(* IEC 61131-3 sources: Industry-PLC-LLM/data/PLCBEAD_repo/PLCBEAD_PLCEmbed-main/PLC-BEAD/Source/OpenPLCv2 (part 11) *)

(* ---- CEIL2.ST ---- *)
FUNCTION _REAL_TO_DINT:DINT
  VAR_INPUT
    X :	REAL;
  END_VAR

  IF REAL_TO_DINT(0.5) = DINT#1 THEN
    _REAL_TO_DINT := REAL_TO_DINT(x);
    RETURN;
  END_IF;

  IF X > 0.0 THEN
    _REAL_TO_DINT := REAL_TO_DINT(x+0.5);
  ELSIF X < 0.0 THEN
    _REAL_TO_DINT := REAL_TO_DINT(x-0.5);
  ELSE
    _REAL_TO_DINT := DINT#0;
  END_IF;
END_FUNCTION

FUNCTION CEIL2:DINT

	VAR_INPUT
		X :	REAL;
	END_VAR

	CEIL2 := _REAL_TO_DINT(x);
	IF DINT_TO_REAL(CEIL2) < X THEN
			CEIL2 := CEIL2 + DINT#1;
	END_IF;

END_FUNCTION

PROGRAM program0
  VAR
    LocalVar0 : REAL;
    CEIL5_OUT : DINT;
  END_VAR

  CEIL5_OUT := CEIL2(LocalVar0);
END_PROGRAM

CONFIGURATION Config0

  RESOURCE Res0 ON PLC
    TASK task0(INTERVAL := T#20ms,PRIORITY := 0);
    PROGRAM instance0 WITH task0 : program0;
  END_RESOURCE
END_CONFIGURATION

(* ---- CHECK_PARITY.ST ---- *)
FUNCTION BIT_OF_DWORD : BOOL
  VAR_INPUT
    IN : DWORD;
    N : INT;
  END_VAR

  BIT_OF_DWORD := (SHR(in,N) AND 16#00000001) > 0;
END_FUNCTION

FUNCTION CHECK_PARITY:BOOL

	VAR_INPUT
		IN :	DWORD;
		P :	BOOL;
	END_VAR

	VAR
		in2 :	DWORD;
	END_VAR

	in2:=in;
	check_parity := NOT p;
	WHILE in2 > DWORD#0 DO
		check_parity := check_parity XOR BIT_OF_DWORD(in2,0) XOR BIT_OF_DWORD(in2,1) XOR BIT_OF_DWORD(in2,2) XOR BIT_OF_DWORD(in2,3);
		in2 := SHR(in2,4);
	END_WHILE;

END_FUNCTION

PROGRAM program0
  VAR
    LocalVar0 : DWORD;
    LocalVar1 : BOOL;
    CEIL5_OUT : BOOL;
  END_VAR

  CEIL5_OUT := CHECK_PARITY(LocalVar0, LocalVar1);
END_PROGRAM

CONFIGURATION Config0

  RESOURCE Res0 ON PLC
    TASK task0(INTERVAL := T#20ms,PRIORITY := 0);
    PROGRAM instance0 WITH task0 : program0;
  END_RESOURCE
END_CONFIGURATION

(* ---- CIRCLE_A.ST ---- *)
FUNCTION CIRCLE_A:REAL
	VAR_INPUT
		RX :	REAL;
		AX :	REAL;
	END_VAR

	circle_A := Rx * RX * 8.726646E-3 * Ax;
END_FUNCTION

PROGRAM program0
  VAR
    LocalVar0 : REAL;
	LocalVar1 : REAL;
	LocalOUT  : REAL;
  END_VAR
  	LocalOUT := CIRCLE_A(LocalVar0, LocalVar1);
END_PROGRAM

CONFIGURATION Config0
  RESOURCE Res0 ON PLC
    TASK task0(INTERVAL := T#20ms,PRIORITY := 0);
    PROGRAM instance0 WITH task0 : program0;
  END_RESOURCE
END_CONFIGURATION

(* ---- CIRCLE_C.ST ---- *)
FUNCTION CIRCLE_C:REAL
	VAR_INPUT
		RX :	REAL;
		AX :	REAL;
	END_VAR

	circle_C := 1.7453293E-2 * Rx * Ax;
END_FUNCTION

PROGRAM program0
  VAR
    LocalVar0 : REAL;
	LocalVar1 : REAL;
	LocalOUT  : REAL;
  END_VAR
  	LocalOUT := CIRCLE_C(LocalVar0, LocalVar1);
END_PROGRAM

CONFIGURATION Config0
  RESOURCE Res0 ON PLC
    TASK task0(INTERVAL := T#20ms,PRIORITY := 0);
    PROGRAM instance0 WITH task0 : program0;
  END_RESOURCE
END_CONFIGURATION

(* ---- CIRCLE_SEG.ST ---- *)
FUNCTION CIRCLE_SEG:REAL
	VAR_INPUT
		RX :	REAL;
		HX :	REAL;
	END_VAR

	IF RX > 0.0 THEN
		CIRCLE_SEG := 2.0 * ACOS(1.0 - LIMIT(0.0, HX / RX, 2.0));
		CIRCLE_SEG := (CIRCLE_SEG - SIN(CIRCLE_SEG)) * RX * RX * 0.5;
	END_IF;
END_FUNCTION

PROGRAM program0
  VAR
    LocalVar0 : REAL;
	LocalVar1 : REAL;
	LocalOUT  : REAL;
  END_VAR
  	LocalOUT := CIRCLE_SEG(LocalVar0, LocalVar1);
END_PROGRAM

CONFIGURATION Config0
  RESOURCE Res0 ON PLC
    TASK task0(INTERVAL := T#20ms,PRIORITY := 0);
    PROGRAM instance0 WITH task0 : program0;
  END_RESOURCE
END_CONFIGURATION

(* ---- CMP.ST ---- *)
FUNCTION EXP10 : REAL
  VAR_INPUT
    x : REAL;
  END_VAR

  exp10 := EXP(X * 2.30258509299405);
  (* from OSCAT library; www.oscat.de  *)
END_FUNCTION

FUNCTION FLOOR : INT
  VAR_INPUT
    x : REAL;
  END_VAR

  FLOOR := REAL_TO_INT(X);
  IF INT_TO_REAL(FLOOR) > X THEN
  	floor := floor - 1;
  END_IF;
  (* from OSCAT library; www.oscat.de  *)
END_FUNCTION

FUNCTION CMP:BOOL
	VAR_INPUT
		X :	REAL;
		Y :	REAL;
		N :	INT;
	END_VAR

	VAR
		tmp :	REAL;
	END_VAR

	tmp := ABS(x);
	IF tmp > 0.0 THEN
		tmp := EXP10(INT_TO_REAL(FLOOR(LOG(tmp))-N+1));
	ELSE
		tmp := EXP10(tmp);
	END_IF;
	CMP := ABS(X - Y) < tmp;

END_FUNCTION

PROGRAM program0
  VAR
    LocalVar0 : REAL;
    LocalVar1 : REAL;
	LocalVar2 : INT;
    CEIL5_OUT : BOOL;
  END_VAR

  CEIL5_OUT := CMP(LocalVar0, LocalVar1, LocalVar2);
END_PROGRAM

CONFIGURATION Config0

  RESOURCE Res0 ON PLC
    TASK task0(INTERVAL := T#20ms,PRIORITY := 0);
    PROGRAM instance0 WITH task0 : program0;
  END_RESOURCE
END_CONFIGURATION

(* ---- CONE_V.ST ---- *)
FUNCTION CONE_V:REAL
	VAR_INPUT
		RX :	REAL;
		HX :	REAL;
	END_VAR

	cone_V := 1.047197551 * RX * RX * hx;
END_FUNCTION

PROGRAM program0
  VAR
    LocalVar0 : REAL;
	LocalVar1 : REAL;
	LocalOUT  : REAL;
  END_VAR
  	LocalOUT := CONE_V(LocalVar0, LocalVar1);
END_PROGRAM

CONFIGURATION Config0
  RESOURCE Res0 ON PLC
    TASK task0(INTERVAL := T#20ms,PRIORITY := 0);
    PROGRAM instance0 WITH task0 : program0;
  END_RESOURCE
END_CONFIGURATION

(* ---- COSH.ST ---- *)
FUNCTION COSH:REAL
	VAR_INPUT
		X :	REAL;
	END_VAR

	VAR
		t :	REAL;
	END_VAR

	T := EXP(X);
	COSH := (1.0 / T + T) * 0.5;
END_FUNCTION

PROGRAM program0
  VAR
    LocalVar0 : REAL;
    CEIL5_OUT : REAL;
  END_VAR

  CEIL5_OUT := COSH(LocalVar0);
END_PROGRAM

CONFIGURATION Config0

  RESOURCE Res0 ON PLC
    TASK task0(INTERVAL := T#20ms,PRIORITY := 0);
    PROGRAM instance0 WITH task0 : program0;
  END_RESOURCE
END_CONFIGURATION

(* ---- COTH.ST ---- *)
FUNCTION COTH:REAL

	VAR_INPUT
		X :	REAL;
	END_VAR

	IF X > 20.0 THEN
		COTH :=1.0;
	ELSIF X < -20.0 THEN
		COTH := -1.0;
	ELSE
		COTH := 1.0 + 2.0 / (EXP(X * 2.0) - 1.0);
	END_IF;

END_FUNCTION

PROGRAM program0
	VAR
		X :	REAL;
		OUT : REAL;
	END_VAR

	OUT := COTH(X);

END_PROGRAM

CONFIGURATION Config0

	RESOURCE Res0 ON PLC
		TASK task0(INTERVAL := T#20ms,PRIORITY := 0);
		PROGRAM instance0 WITH task0 : program0;
	END_RESOURCE

END_CONFIGURATION

(* ---- CTRL_IN.ST ---- *)
FUNCTION DEAD_ZONE:REAL

	VAR_INPUT
		X :	REAL;
		L :	REAL;
	END_VAR

	IF ABS(x) > L THEN
		dead_zone := X;
	ELSE
		DEAD_ZONE := 0.0;
	END_IF;

END_FUNCTION

FUNCTION CTRL_IN:REAL
	VAR_INPUT
		SET_POINT :	REAL;
		ACTUAL :	REAL;
		NOISE :	REAL;
	END_VAR
	CTRL_IN := DEAD_ZONE(SET_POINT - ACTUAL, NOISE);
END_FUNCTION

PROGRAM program0
  VAR
    LocalVar0 : REAL;
	LocalVar1 : REAL;
	LocalVar2 : REAL;
	LocalOUT  : REAL;
  END_VAR
  	LocalOUT := CTRL_IN(LocalVar0, LocalVar1, LocalVar2);
END_PROGRAM

CONFIGURATION Config0
  RESOURCE Res0 ON PLC
    TASK task0(INTERVAL := T#20ms,PRIORITY := 0);
    PROGRAM instance0 WITH task0 : program0;
  END_RESOURCE
END_CONFIGURATION

(* ---- D_TRUNC.ST ---- *)
FUNCTION D_TRUNC : DINT
  VAR_INPUT
    x : REAL;
  END_VAR

  D_TRUNC := REAL_TO_DINT(X);
  IF X > 0.0 THEN
  	IF DINT_TO_REAL(D_TRUNC) > X THEN D_TRUNC := D_TRUNC - DINT#1; END_IF;
  ELSE
  	IF DINT_TO_REAL(D_TRUNC) < X THEN D_TRUNC := D_TRUNC + DINT#1; END_IF;
  END_IF;
END_FUNCTION

PROGRAM program0
  VAR
    LocalVar0 : REAL;
    LocalVar1 : DINT;
    CEIL5_OUT : DINT;
  END_VAR

  CEIL5_OUT := D_TRUNC(LocalVar0);
  LocalVar1 := CEIL5_OUT;
END_PROGRAM

CONFIGURATION Config0

  RESOURCE Res0 ON PLC
    TASK task0(INTERVAL := T#20ms,PRIORITY := 0);
    PROGRAM instance0 WITH task0 : program0;
  END_RESOURCE
END_CONFIGURATION

(* ---- DATE_ADD.ST ---- *)
FUNCTION YEAR_OF_DATE:INT
	VAR_INPUT
		IDATE :	UDINT;
	END_VAR

	YEAR_OF_DATE := UDINT_TO_INT((idate+UDINT#43200) / UDINT#31557600 + UDINT#1970);
END_FUNCTION

FUNCTION DAY_OF_WEEK:INT

	VAR_INPUT
		IDATE :	UDINT;
	END_VAR

	DAY_OF_WEEK := UDINT_TO_INT((idate / UDINT#86400 + UDINT#3) MOD UDINT#7) + INT#01;
END_FUNCTION

FUNCTION LEAP_OF_DATE:BOOL

	VAR_INPUT
		IDATE :	UDINT;
	END_VAR

	LEAP_OF_DATE := SHL(UDINT_TO_DWORD((idate + UDINT#43200) / UDINT#31557600), 30) = DWORD#16#80000000;
END_FUNCTION

FUNCTION DAY_OF_YEAR:INT
	VAR_INPUT
		IDATE :	UDINT;
	END_VAR

	DAY_OF_YEAR := UDINT_TO_INT(((idate) / UDINT#86400) MOD UDINT#1461);
	IF DAY_OF_YEAR > 729 THEN
		IF DAY_OF_YEAR > 1095 THEN DAY_OF_YEAR := DAY_OF_YEAR - 1095; ELSE DAY_OF_YEAR := DAY_OF_YEAR - 729; END_IF;
	ELSIF DAY_OF_YEAR > 364 THEN
		DAY_OF_YEAR := DAY_OF_YEAR - 364;
	ELSE
		DAY_OF_YEAR := DAY_OF_YEAR + 1;
	END_IF;
END_FUNCTION

FUNCTION MONTH_OF_DATE:INT

	VAR_INPUT
		IDATE :	UDINT;
	END_VAR

	MONTH_OF_DATE := DAY_OF_YEAR(idate);
	IF MONTH_OF_DATE < 32 THEN
		MONTH_OF_DATE := 1;
	ELSIF LEAP_OF_DATE((IDATE)) THEN
		MONTH_OF_DATE := (MONTH_OF_DATE * 53 + 1668) / 1623;
	ELSE
		MONTH_OF_DATE := (MONTH_OF_DATE * 53 + 1700) / 1620;
	END_IF;
END_FUNCTION

FUNCTION DAY_OF_MONTH:INT
	VAR_INPUT
		IDATE :	UDINT;
	END_VAR

	day_of_month := day_of_year(idate);

	IF leap_of_Date((idate)) THEN
		CASE day_of_month OF
			32..60	:	day_of_month := day_of_month - 31;
			61..91	:	day_of_month := day_of_month - 60;
			92..121 :	day_of_month := day_of_month - 91;
			122..152:	day_of_month := day_of_month - 121;
			153..182:	day_of_month := day_of_month - 152;
			183..213:	day_of_month := day_of_month - 182;
			214..244:	day_of_month := day_of_month - 213;
			245..274:	day_of_month := day_of_month - 244;
			275..305:	day_of_month := day_of_month - 274;
			306..335:	day_of_month := day_of_month - 305;
			336..366:	day_of_month := day_of_month - 335;
		END_CASE;
	ELSE
		CASE day_of_month OF
			32..59	:	day_of_month := day_of_month - 31;
			60..90	:	day_of_month := day_of_month - 59;
			91..120 :	day_of_month := day_of_month - 90;
			121..151:	day_of_month := day_of_month - 120;
			152..181:	day_of_month := day_of_month - 151;
			182..212:	day_of_month := day_of_month - 181;
			213..243:	day_of_month := day_of_month - 212;
			244..273:	day_of_month := day_of_month - 243;
			274..304:	day_of_month := day_of_month - 273;
			305..334:	day_of_month := day_of_month - 304;
			335..365:	day_of_month := day_of_month - 334;
		END_CASE;
	END_IF;
END_FUNCTION

FUNCTION _INT_TO_UDINT:UDINT
	VAR_INPUT
		IN :	INT;
	END_VAR

	_INT_TO_UDINT := DINT_TO_UDINT(INT_TO_DINT(IN));
END_FUNCTION

FUNCTION SET_DATE:UDINT

	VAR_INPUT
		YEAR :	INT;
		MONTH :	INT;
		DAY :	INT;
	END_VAR

	VAR
		count :	INT;
	END_VAR

	IF month > 2 THEN
		count := (month - 1) * 30;
		IF month > 7 THEN
			count := count + DWORD_TO_INT(SHR(DINT_TO_DWORD(INT_TO_DINT(month) - INT_TO_DINT(3)),1));
		ELSE
			count := count + DWORD_TO_INT(SHR(DINT_TO_DWORD(INT_TO_DINT(month) - INT_TO_DINT(4)),1));
		END_IF;
		IF SHL(INT_TO_WORD(year),14) = WORD#0 THEN
			count := count + 1;
		END_IF;
	ELSE
		count := (month - 1) * 31;
	END_IF;
	SET_DATE := (_INT_TO_UDINT(count + day - 1) + DWORD_TO_UDINT(SHR(UDINT_TO_DWORD(_INT_TO_UDINT(year) * UDINT#1461 - UDINT#2878169), 2))) * UDINT#86400;

END_FUNCTION

FUNCTION DATE_ADD:UDINT
	VAR_INPUT
		IDATE :	UDINT;
		D :	INT;
		W :	INT;
		M :	INT;
		Y :	INT;
	END_VAR

	VAR
		mo :	INT;
		yr :	INT;
		dm :	INT;
	END_VAR

	DATE_ADD := IDATE + INT_TO_UDINT(D + W * 7) * UDINT#86400;
	yr := Y + YEAR_OF_DATE(DATE_ADD);
	mo := M + MONTH_OF_DATE(DATE_ADD);
	dm := DAY_OF_MONTH(DATE_ADD);
	WHILE mo > 12 DO
		mo := mo - 12;
		yr := yr + 1;
	END_WHILE;
	WHILE mo < 1 DO
		mo := mo + 12;
		yr := yr - 1;
	END_WHILE;
	DATE_ADD := SET_DATE(yr, mo, dm);
END_FUNCTION

PROGRAM program0
  VAR
    LocalVar0 : UDINT;
	LocalVar1 : INT;
	LocalVar2 : INT;
	LocalVar3 : INT;
	LocalVar4 : INT;
	LocalOUT  : UDINT;
  END_VAR
  	LocalOUT := DATE_ADD(LocalVar0, LocalVar1, LocalVar2, LocalVar3, LocalVar4);
END_PROGRAM

CONFIGURATION Config0
  RESOURCE Res0 ON PLC
    TASK task0(INTERVAL := T#20ms,PRIORITY := 0);
    PROGRAM instance0 WITH task0 : program0;
  END_RESOURCE
END_CONFIGURATION

(* ---- DATE_TO_DT.ST ---- *)
FUNCTION DATE_TO_DT:UDINT
	VAR_INPUT
		IN :	UDINT;
	END_VAR
	DATE_TO_DT := IN;
END_FUNCTION

PROGRAM program0
  VAR
    LocalVar0 : UDINT;
	LocalOUT  : UDINT;
  END_VAR
  	LocalOUT := DATE_TO_DT(LocalVar0);
END_PROGRAM

CONFIGURATION Config0
  RESOURCE Res0 ON PLC
    TASK task0(INTERVAL := T#20ms,PRIORITY := 0);
    PROGRAM instance0 WITH task0 : program0;
  END_RESOURCE
END_CONFIGURATION

(* ---- DATE_TO_DWORD.ST ---- *)
FUNCTION DATE_TO_DWORD2:DWORD
	VAR_INPUT
		IN :	UDINT;
	END_VAR

	DATE_TO_DWORD2 := UDINT_TO_DWORD(IN);
END_FUNCTION

PROGRAM program0
  VAR
    LocalVar0 : UDINT;
	LocalOUT  : DWORD;
  END_VAR
  	LocalOUT := DATE_TO_DWORD2(LocalVar0);
END_PROGRAM

CONFIGURATION Config0
  RESOURCE Res0 ON PLC
    TASK task0(INTERVAL := T#20ms,PRIORITY := 0);
    PROGRAM instance0 WITH task0 : program0;
  END_RESOURCE
END_CONFIGURATION

(* ---- DATE_TO_REAL.ST ---- *)
FUNCTION DATE_TO_REAL2:REAL
	VAR_INPUT
		IN :	UDINT;
	END_VAR

	DATE_TO_REAL2 := UDINT_TO_REAL(IN);
END_FUNCTION

PROGRAM program0
  VAR
    LocalVar0 : UDINT;
	LocalOUT  : REAL;
  END_VAR
  	LocalOUT := DATE_TO_REAL2(LocalVar0);
END_PROGRAM

CONFIGURATION Config0
  RESOURCE Res0 ON PLC
    TASK task0(INTERVAL := T#20ms,PRIORITY := 0);
    PROGRAM instance0 WITH task0 : program0;
  END_RESOURCE
END_CONFIGURATION

(* ---- DATE_TO_UDINT.ST ---- *)
FUNCTION DATE_TO_UDINT2:UDINT
	VAR_INPUT
		IN :	UDINT;
	END_VAR

	DATE_TO_UDINT2 := IN;
END_FUNCTION

PROGRAM program0
  VAR
    LocalVar0 : UDINT;
	LocalOUT  : UDINT;
  END_VAR
  	LocalOUT := DATE_TO_UDINT2(LocalVar0);
END_PROGRAM

CONFIGURATION Config0
  RESOURCE Res0 ON PLC
    TASK task0(INTERVAL := T#20ms,PRIORITY := 0);
    PROGRAM instance0 WITH task0 : program0;
  END_RESOURCE
END_CONFIGURATION

(* ---- DAY_OF_DATE.ST ---- *)
FUNCTION DAY_OF_DATE:DINT
	VAR_INPUT
		IDATE :	UDINT;
	END_VAR

	day_of_date := UDINT_TO_DINT(idate / UDINT#86400);
END_FUNCTION

PROGRAM program0
  VAR
    LocalVar0 : UDINT;
	LocalOUT  : DINT;
  END_VAR
  	LocalOUT := DAY_OF_DATE(LocalVar0);
END_PROGRAM

CONFIGURATION Config0
  RESOURCE Res0 ON PLC
    TASK task0(INTERVAL := T#20ms,PRIORITY := 0);
    PROGRAM instance0 WITH task0 : program0;
  END_RESOURCE
END_CONFIGURATION

(* ---- DAY_OF_MONTH.ST ---- *)
FUNCTION LEAP_OF_DATE:BOOL

	VAR_INPUT
		IDATE :	UDINT;
	END_VAR

	LEAP_OF_DATE := SHL(UDINT_TO_DWORD((idate + UDINT#43200) / UDINT#31557600), 30) = DWORD#16#80000000;

END_FUNCTION

FUNCTION DAY_OF_YEAR:INT
	VAR_INPUT
		IDATE :	DATE;
	END_VAR

	DAY_OF_YEAR := UDINT_TO_INT((DATE_TO_UDINT(idate) / UDINT#86400) MOD UDINT#1461);
	IF DAY_OF_YEAR > 729 THEN
		IF DAY_OF_YEAR > 1095 THEN DAY_OF_YEAR := DAY_OF_YEAR - 1095; ELSE DAY_OF_YEAR := DAY_OF_YEAR - 729; END_IF;
	ELSIF DAY_OF_YEAR > 364 THEN
		DAY_OF_YEAR := DAY_OF_YEAR - 364;
	ELSE
		DAY_OF_YEAR := DAY_OF_YEAR + 1;
	END_IF;
END_FUNCTION

FUNCTION DAY_OF_MONTH:INT
	VAR_INPUT
		IDATE :	DATE;
	END_VAR

	day_of_month := day_of_year(idate);

	IF leap_of_Date(DATE_TO_UDINT(idate)) THEN
		CASE day_of_month OF
			32..60	:	day_of_month := day_of_month - 31;
			61..91	:	day_of_month := day_of_month - 60;
			92..121 :	day_of_month := day_of_month - 91;
			122..152:	day_of_month := day_of_month - 121;
			153..182:	day_of_month := day_of_month - 152;
			183..213:	day_of_month := day_of_month - 182;
			214..244:	day_of_month := day_of_month - 213;
			245..274:	day_of_month := day_of_month - 244;
			275..305:	day_of_month := day_of_month - 274;
			306..335:	day_of_month := day_of_month - 305;
			336..366:	day_of_month := day_of_month - 335;
		END_CASE;
	ELSE
		CASE day_of_month OF
			32..59	:	day_of_month := day_of_month - 31;
			60..90	:	day_of_month := day_of_month - 59;
			91..120 :	day_of_month := day_of_month - 90;
			121..151:	day_of_month := day_of_month - 120;
			152..181:	day_of_month := day_of_month - 151;
			182..212:	day_of_month := day_of_month - 181;
			213..243:	day_of_month := day_of_month - 212;
			244..273:	day_of_month := day_of_month - 243;
			274..304:	day_of_month := day_of_month - 273;
			305..334:	day_of_month := day_of_month - 304;
			335..365:	day_of_month := day_of_month - 334;
		END_CASE;
	END_IF;

END_FUNCTION

PROGRAM program0
  VAR
    LocalVar0 : DATE;
	LocalOUT  : INT;
  END_VAR
  	LocalOUT := DAY_OF_MONTH(LocalVar0);
END_PROGRAM

CONFIGURATION Config0
  RESOURCE Res0 ON PLC
    TASK task0(INTERVAL := T#20ms,PRIORITY := 0);
    PROGRAM instance0 WITH task0 : program0;
  END_RESOURCE
END_CONFIGURATION

(* ---- DAY_OF_WEEK.ST ---- *)
FUNCTION DAY_OF_WEEK:INT
  VAR_INPUT
    IDATE :	UDINT;
  END_VAR

  DAY_OF_WEEK := UDINT_TO_INT((idate / UDINT#86400 + UDINT#3) MOD UDINT#7) + INT#01;
END_FUNCTION

PROGRAM program0
  VAR
    LocalVar0 : UDINT;
	LocalOUT  : INT;
  END_VAR
  	LocalOUT := DAY_OF_WEEK(LocalVar0);
END_PROGRAM

CONFIGURATION Config0
  RESOURCE Res0 ON PLC
    TASK task0(INTERVAL := T#20ms,PRIORITY := 0);
    PROGRAM instance0 WITH task0 : program0;
  END_RESOURCE
END_CONFIGURATION

(* ---- DAY_OF_YEAR.ST ---- *)
FUNCTION DAY_OF_YEAR:INT
	VAR_INPUT
		IDATE :	DATE;
	END_VAR

	DAY_OF_YEAR := UDINT_TO_INT((DATE_TO_UDINT(idate) / UDINT#86400) MOD UDINT#1461);
	IF DAY_OF_YEAR > 729 THEN
		IF DAY_OF_YEAR > 1095 THEN DAY_OF_YEAR := DAY_OF_YEAR - 1095; ELSE DAY_OF_YEAR := DAY_OF_YEAR - 729; END_IF;
	ELSIF DAY_OF_YEAR > 364 THEN
		DAY_OF_YEAR := DAY_OF_YEAR - 364;
	ELSE
		DAY_OF_YEAR := DAY_OF_YEAR + 1;
	END_IF;
END_FUNCTION

PROGRAM program0
  VAR
    LocalVar0 : DATE;
	LocalOUT  : INT;
  END_VAR
  	LocalOUT := DAY_OF_YEAR(LocalVar0);
END_PROGRAM

CONFIGURATION Config0
  RESOURCE Res0 ON PLC
    TASK task0(INTERVAL := T#20ms,PRIORITY := 0);
    PROGRAM instance0 WITH task0 : program0;
  END_RESOURCE
END_CONFIGURATION

(* ---- DAYS_DELTA.ST ---- *)
FUNCTION DAYS_DELTA:DINT
	VAR_INPUT
		DATE_1 :	UDINT;
		DATE_2 :	UDINT;
	END_VAR
	IF DATE_1 > DATE_2 THEN
		DAYS_DELTA := - UDINT_TO_DINT((date_1 - date_2) / UDINT#86400);
	ELSE
		DAYS_DELTA :=   UDINT_TO_DINT((date_2 - date_1) / UDINT#86400);
	END_IF;
END_FUNCTION

PROGRAM program0
  VAR
    LocalVar0 : UDINT;
	LocalVar1 : UDINT;
	LocalOUT  : DINT;
  END_VAR
  	LocalOUT := DAYS_DELTA(LocalVar0, LocalVar1);
END_PROGRAM

CONFIGURATION Config0
  RESOURCE Res0 ON PLC
    TASK task0(INTERVAL := T#20ms,PRIORITY := 0);
    PROGRAM instance0 WITH task0 : program0;
  END_RESOURCE
END_CONFIGURATION

(* ---- DAYS_IN_MONTH.ST ---- *)
FUNCTION DAY_OF_YEAR:INT
	VAR_INPUT
		IDATE :	UDINT;
	END_VAR

	DAY_OF_YEAR := UDINT_TO_INT(((idate) / UDINT#86400) MOD UDINT#1461);
	IF DAY_OF_YEAR > 729 THEN
		IF DAY_OF_YEAR > 1095 THEN DAY_OF_YEAR := DAY_OF_YEAR - 1095; ELSE DAY_OF_YEAR := DAY_OF_YEAR - 729; END_IF;
	ELSIF DAY_OF_YEAR > 364 THEN
		DAY_OF_YEAR := DAY_OF_YEAR - 364;
	ELSE
		DAY_OF_YEAR := DAY_OF_YEAR + 1;
	END_IF;
END_FUNCTION

FUNCTION LEAP_OF_DATE:BOOL

	VAR_INPUT
		IDATE :	UDINT;
	END_VAR

	LEAP_OF_DATE := SHL(UDINT_TO_DWORD((idate + UDINT#43200) / UDINT#31557600), 30) = DWORD#16#80000000;
END_FUNCTION

FUNCTION DAYS_IN_MONTH:INT

	VAR_INPUT
		IDATE :	UDINT;
	END_VAR

	DAYS_IN_MONTH := DAY_OF_YEAR(IDATE);
	IF LEAP_OF_DATE(IDATE) THEN
		CASE DAYS_IN_MONTH OF
			32..60	:	DAYS_IN_MONTH := 29;
			92..121 :	DAYS_IN_MONTH := 30;
			153..182:	DAYS_IN_MONTH := 30;
			245..274:	DAYS_IN_MONTH := 30;
			306..335:	DAYS_IN_MONTH := 30;
		ELSE
			DAYS_IN_MONTH := 31;
		END_CASE;
	ELSE
		CASE DAYS_IN_MONTH OF
			32..59	:	DAYS_IN_MONTH := 28;
			91..120 :	DAYS_IN_MONTH := 30;
			152..181:	DAYS_IN_MONTH := 30;
			244..273:	DAYS_IN_MONTH := 30;
			305..334:	DAYS_IN_MONTH := 30;
		ELSE
			DAYS_IN_MONTH := 31;
		END_CASE;
	END_IF;

END_FUNCTION

PROGRAM program0
  VAR
    LocalVar0 : UDINT;
	LocalOUT  : INT;
  END_VAR
  	LocalOUT := DAYS_IN_MONTH(LocalVar0);
END_PROGRAM

CONFIGURATION Config0
  RESOURCE Res0 ON PLC
    TASK task0(INTERVAL := T#20ms,PRIORITY := 0);
    PROGRAM instance0 WITH task0 : program0;
  END_RESOURCE
END_CONFIGURATION

(* ---- DAYS_IN_YEAR.ST ---- *)
FUNCTION LEAP_OF_DATE:BOOL

	VAR_INPUT
		IDATE :	UDINT;
	END_VAR

	LEAP_OF_DATE := SHL(UDINT_TO_DWORD((idate + UDINT#43200) / UDINT#31557600), 30) = DWORD#16#80000000;
END_FUNCTION

FUNCTION DAYS_IN_YEAR:INT
	VAR_INPUT
		IDATE :	UDINT;
	END_VAR

	IF LEAP_OF_DATE(IDATE) THEN
		DAYS_IN_YEAR := 366;
	ELSE
		DAYS_IN_YEAR := 365;
	END_IF;
END_FUNCTION

PROGRAM program0
  VAR
    LocalVar0 : UDINT;
	LocalOUT  : INT;
  END_VAR
  	LocalOUT := DAYS_IN_YEAR(LocalVar0);
END_PROGRAM

CONFIGURATION Config0
  RESOURCE Res0 ON PLC
    TASK task0(INTERVAL := T#20ms,PRIORITY := 0);
    PROGRAM instance0 WITH task0 : program0;
  END_RESOURCE
END_CONFIGURATION

(* ---- DEAD_BAND.ST ---- *)
FUNCTION DEAD_BAND:REAL

	VAR_INPUT
		X :	REAL;
		L :	REAL;
	END_VAR

	IF X > L THEN
		DEAD_BAND := X - L;
	ELSIF X < -L THEN
		DEAD_BAND := X + L;
	ELSE
		DEAD_BAND := 0.0;
	END_IF;

END_FUNCTION

PROGRAM program0
  VAR
    LocalVar0 : REAL;
	LocalVar1 : REAL;
	LocalOUT  : REAL;
  END_VAR
  	LocalOUT := DEAD_BAND(LocalVar0, LocalVar1);
END_PROGRAM

CONFIGURATION Config0
  RESOURCE Res0 ON PLC
    TASK task0(INTERVAL := T#20ms,PRIORITY := 0);
    PROGRAM instance0 WITH task0 : program0;
  END_RESOURCE
END_CONFIGURATION

(* ---- DEAD_ZONE.ST ---- *)
FUNCTION DEAD_ZONE:REAL

	VAR_INPUT
		X :	REAL;
		L :	REAL;
	END_VAR

	IF ABS(x) > L THEN
		dead_zone := X;
	ELSE
		DEAD_ZONE := 0.0;
	END_IF;

END_FUNCTION

PROGRAM program0
  VAR
    LocalVar0 : REAL;
	LocalVar1 : REAL;
	LocalOUT  : REAL;
  END_VAR
  	LocalOUT := DEAD_ZONE(LocalVar0, LocalVar1);
END_PROGRAM

CONFIGURATION Config0
  RESOURCE Res0 ON PLC
    TASK task0(INTERVAL := T#20ms,PRIORITY := 0);
    PROGRAM instance0 WITH task0 : program0;
  END_RESOURCE
END_CONFIGURATION

(* ---- DEC1.ST ---- *)
FUNCTION DEC1:INT

	VAR_INPUT
		X :	INT;
		N :	INT;
	END_VAR

	IF X = 0 THEN
		DEC1 := N - 1;
	ELSE
		DEC1 := X - 1;
	END_IF;

END_FUNCTION

PROGRAM program0
  VAR
    LocalVar0 : INT;
	LocalVar1 : INT;
	LocalOUT  : INT;
  END_VAR
  	LocalOUT := DEC1(LocalVar0, LocalVar1);
END_PROGRAM

CONFIGURATION Config0
  RESOURCE Res0 ON PLC
    TASK task0(INTERVAL := T#20ms,PRIORITY := 0);
    PROGRAM instance0 WITH task0 : program0;
  END_RESOURCE
END_CONFIGURATION

(* ---- DEG.ST ---- *)
FUNCTION FLOOR2 : DINT
	VAR_INPUT
		x : REAL;
	END_VAR

	FLOOR2 := REAL_TO_DINT(X);
	IF DINT_TO_REAL(FLOOR2) > X THEN
		FLOOR2 := FLOOR2 - DINT#1;
	END_IF;

END_FUNCTION

FUNCTION MODR:REAL

	VAR_INPUT
		IN :	REAL;
		DIVI :	REAL;
	END_VAR

	IF divi = 0.0 THEN
		MODR := 0.0;
	ELSE
		MODR := in - DINT_TO_REAL(FLOOR2(in / divi)) * divi;
	END_IF;

END_FUNCTION

FUNCTION DEG:REAL

	VAR_INPUT
		RAD :	REAL;
	END_VAR

	DEG := MODR(57.29577951308232 * RAD, 360.0);

END_FUNCTION

PROGRAM program0

	VAR
		RAD :	REAL;
		CEIL5_OUT : REAL;
	END_VAR

	CEIL5_OUT := DEG(RAD);

END_PROGRAM

CONFIGURATION Config0

	RESOURCE Res0 ON PLC
		TASK task0(INTERVAL := T#20ms,PRIORITY := 0);
		PROGRAM instance0 WITH task0 : program0;
	END_RESOURCE

END_CONFIGURATION

(* ---- DEW_CON.ST ---- *)
FUNCTION SDD:REAL

	VAR_INPUT
		T :	REAL;
		ICE :	BOOL;
	END_VAR

	IF ice THEN
		SDD := 611.153 * EXP(22.4433 * T / (272.186 + T));
	ELSE
		SDD := 611.213 * EXP(17.5043 * T / (241.2 + T));
	END_IF;

END_FUNCTION

FUNCTION DEW_CON:REAL

	VAR_INPUT
		RH :	REAL;
		T :	REAL;
	END_VAR

	IF RH > 0.0 AND T > -50.0 THEN
		DEW_CON := 2.166824303E-2 * RH * SDD(T,FALSE)  / (T - -273.15);
	ELSE
		DEW_CON := 0.0;
	END_IF;

END_FUNCTION

PROGRAM program0
  VAR
    RH :	REAL;
	T :	REAL;
    CEIL5_OUT : REAL;
  END_VAR

  CEIL5_OUT := DEW_CON(RH, T);
END_PROGRAM

CONFIGURATION Config0

  RESOURCE Res0 ON PLC
    TASK task0(INTERVAL := T#20ms,PRIORITY := 0);
    PROGRAM instance0 WITH task0 : program0;
  END_RESOURCE
END_CONFIGURATION

(* ---- DEW_RH.ST ---- *)
FUNCTION SDD:REAL

	VAR_INPUT
		T :	REAL;
		ICE :	BOOL;
	END_VAR

	IF ice THEN
		SDD := 611.153 * EXP(22.4433 * T / (272.186 + T));
	ELSE
		SDD := 611.213 * EXP(17.5043 * T / (241.2 + T));
	END_IF;

END_FUNCTION

FUNCTION DEW_CON:REAL

	VAR_INPUT
		RH :	REAL;
		T :	REAL;
	END_VAR

	IF RH > 0.0 AND T > -50.0 THEN
		DEW_CON := 2.166824303E-2 * RH * SDD(T,FALSE)  / (T - -273.15);
	ELSE
		DEW_CON := 0.0;
	END_IF;

END_FUNCTION

FUNCTION DEW_RH:REAL

	VAR_INPUT
		VC :	REAL;
		T :	REAL;
	END_VAR

	DEW_RH := LIMIT(0.0, VC / DEW_CON(1.0, T), 100.0);

END_FUNCTION

PROGRAM program0
	VAR
		VC :	REAL;
		T :	REAL;
		CEIL5_OUT : REAL;
	END_VAR

  	CEIL5_OUT := DEW_RH(VC, T);
END_PROGRAM

CONFIGURATION Config0

  RESOURCE Res0 ON PLC
    TASK task0(INTERVAL := T#20ms,PRIORITY := 0);
    PROGRAM instance0 WITH task0 : program0;
  END_RESOURCE
END_CONFIGURATION

(* ---- DEW_TEMP.ST ---- *)
FUNCTION EXP10 : REAL
  VAR_INPUT
    x : REAL;
  END_VAR

  exp10 := EXP(X * 2.30258509299405);
  (* from OSCAT library; www.oscat.de  *)
END_FUNCTION

FUNCTION DEW_TEMP:REAL

VAR_INPUT
	RH :	REAL;
	T :	REAL;
END_VAR

	VAR
		V :	REAL;
	END_VAR

	IF rh > 0.0 THEN

		V := LOG(RH * 0.01 * EXP10((7.5*T) / (237.3+T)));
		DEW_TEMP := 237.3*V / (7.5-V);
	ELSE
		DEW_TEMP:= -273.15;
	END_IF;

END_FUNCTION

PROGRAM program0
	VAR
		RH :	REAL;
		T :	REAL;
		CEIL5_OUT : REAL;
	END_VAR

  	CEIL5_OUT := DEW_TEMP(RH, T);
END_PROGRAM

CONFIGURATION Config0

  RESOURCE Res0 ON PLC
    TASK task0(INTERVAL := T#20ms,PRIORITY := 0);
    PROGRAM instance0 WITH task0 : program0;
  END_RESOURCE
END_CONFIGURATION

(* ---- DIFFER.ST ---- *)
FUNCTION DIFFER:BOOL
	VAR_INPUT
		IN1 :	REAL;
		IN2 :	REAL;
		X :	REAL;
	END_VAR

	DIFFER := ABS(in1 - in2) > X;
END_FUNCTION

PROGRAM program0
  VAR
    LocalVar0 : REAL;
	LocalVar1 : REAL;
	LocalVar2 : REAL;
	LocalOUT  : BOOL;
  END_VAR
  	LocalOUT := DIFFER(LocalVar0, LocalVar1, LocalVar2);
END_PROGRAM

CONFIGURATION Config0
  RESOURCE Res0 ON PLC
    TASK task0(INTERVAL := T#20ms,PRIORITY := 0);
    PROGRAM instance0 WITH task0 : program0;
  END_RESOURCE
END_CONFIGURATION

(* ---- DST.ST ---- *)
FUNCTION _INT_TO_UDINT:UDINT
	VAR_INPUT
		IN :	INT;
	END_VAR

	_INT_TO_UDINT := DINT_TO_UDINT(INT_TO_DINT(IN));
END_FUNCTION

FUNCTION YEAR_OF_DATE:INT
	VAR_INPUT
		IDATE :	UDINT;
	END_VAR

	YEAR_OF_DATE := UDINT_TO_INT((idate+UDINT#43200) / UDINT#31557600 + UDINT#1970);
END_FUNCTION

FUNCTION DT_TO_DATE2:UDINT

	VAR_INPUT
		IN :	UDINT;
	END_VAR

	DT_TO_DATE2 := (IN / UDINT#86400) * UDINT#86400;
END_FUNCTION

FUNCTION SET_DATE:UDINT

	VAR_INPUT
		YEAR :	INT;
		MONTH :	INT;
		DAY :	INT;
	END_VAR

	VAR
		count :	INT;
	END_VAR

	IF month > 2 THEN
		count := (month - 1) * 30;
		IF month > 7 THEN
			count := count + DWORD_TO_INT(SHR(DINT_TO_DWORD(INT_TO_DINT(month) - INT_TO_DINT(3)),1));
		ELSE
			count := count + DWORD_TO_INT(SHR(DINT_TO_DWORD(INT_TO_DINT(month) - INT_TO_DINT(4)),1));
		END_IF;
		IF SHL(INT_TO_WORD(year),14) = WORD#0 THEN
			count := count + 1;
		END_IF;
	ELSE
		count := (month - 1) * 31;
	END_IF;
	SET_DATE := (_INT_TO_UDINT(count + day - 1) + DWORD_TO_UDINT(SHR(UDINT_TO_DWORD(_INT_TO_UDINT(year) * UDINT#1461 - UDINT#2878169), 2))) * UDINT#86400;

END_FUNCTION

FUNCTION SET_DT:UDINT

	VAR_INPUT
		YEAR :	INT;
		MONTH :	INT;
		DAY :	INT;
		HOUR :	INT;
		MINUTE :	INT;
		SECOND :	INT;
	END_VAR

	SET_DT := SET_DATE(YEAR, MONTH, DAY) + _INT_TO_UDINT(SECOND) + _INT_TO_UDINT(MINUTE) * UDINT#60 + _INT_TO_UDINT(HOUR) * UDINT#3600;

END_FUNCTION

FUNCTION DST:BOOL
	VAR_INPUT
		UTC :	UDINT;
	END_VAR

	VAR
		yr :	INT;
		yr4 :	UDINT;
		ltc :	UDINT;
		idate :	UDINT;
	END_VAR

	yr := YEAR_OF_DATE(DT_TO_DATE2(UTC));
	ltc := UTC;
	idate := SET_DT(yr, 3, 31, 1, 0, 0);
	yr4 := DWORD_TO_UDINT(SHR(INT_TO_DWORD(5 * yr), 2)) + UDINT#1;
	DST := (idate - ((yr4 + UDINT#3) MOD UDINT#7) * UDINT#86400 <= ltc) AND (idate + (UDINT#214 - (yr4) MOD UDINT#7) * UDINT#86400 > ltc);
END_FUNCTION

PROGRAM program0
	VAR
		UTC :	UDINT;
		CEIL5_OUT : BOOL;
	END_VAR

  CEIL5_OUT := DST(UTC);

END_PROGRAM

CONFIGURATION Config0
	RESOURCE Res0 ON PLC
		TASK task0(INTERVAL := T#20ms,PRIORITY := 0);
		PROGRAM instance0 WITH task0 : program0;
	END_RESOURCE
END_CONFIGURATION

(* ---- DT_TO_TOD.ST ---- *)
FUNCTION DT_TO_TOD2:UDINT
	VAR_INPUT
		IN :	UDINT;
	END_VAR

	DT_TO_TOD2 := (IN MOD UDINT#86400) * UDINT#1000;
END_FUNCTION

PROGRAM program0
  VAR
    LocalVar0 : UDINT;
	LocalOUT  : UDINT;
  END_VAR
  	LocalOUT := DT_TO_TOD2(LocalVar0);
END_PROGRAM

CONFIGURATION Config0
  RESOURCE Res0 ON PLC
    TASK task0(INTERVAL := T#20ms,PRIORITY := 0);
    PROGRAM instance0 WITH task0 : program0;
  END_RESOURCE
END_CONFIGURATION

(* ---- DWORD_OF_BYTE.ST ---- *)
FUNCTION DWORD_OF_BYTE:DWORD
	VAR_INPUT
		B3 :	BYTE;
		B2 :	BYTE;
		B1 :	BYTE;
		B0 :	BYTE;
	END_VAR

	DWORD_OF_BYTE := SHL(SHL(SHL(BYTE_TO_DWORD(B3),8) OR BYTE_TO_DWORD(B2),8) OR BYTE_TO_DWORD(B1),8) OR BYTE_TO_DWORD(B0);

END_FUNCTION

PROGRAM program0
  VAR
    LocalVar0 : BYTE;
	LocalVar1 : BYTE;
	LocalVar2 : BYTE;
	LocalVar3 : BYTE;
	LocalOUT  : DWORD;
  END_VAR
  	LocalOUT := DWORD_OF_BYTE(LocalVar0, LocalVar1, LocalVar2, LocalVar3);
END_PROGRAM

CONFIGURATION Config0
  RESOURCE Res0 ON PLC
    TASK task0(INTERVAL := T#20ms,PRIORITY := 0);
    PROGRAM instance0 WITH task0 : program0;
  END_RESOURCE
END_CONFIGURATION

(* ---- DWORD_OF_WORD.ST ---- *)
FUNCTION DWORD_OF_WORD:DWORD

	VAR_INPUT
		W1 :	WORD;
		W0 :	WORD;
	END_VAR

	DWORD_OF_WORD := SHL(WORD_TO_DWORD(W1),16) OR WORD_TO_DWORD(W0);

END_FUNCTION

PROGRAM program0
  VAR
    LocalVar0 : WORD;
	LocalVar1 : WORD;
	LocalOUT  : DWORD;
  END_VAR
  	LocalOUT := DWORD_OF_WORD(LocalVar0, LocalVar1);
END_PROGRAM

CONFIGURATION Config0
  RESOURCE Res0 ON PLC
    TASK task0(INTERVAL := T#20ms,PRIORITY := 0);
    PROGRAM instance0 WITH task0 : program0;
  END_RESOURCE
END_CONFIGURATION

(* ---- DWORD_TO_DATE.ST ---- *)
FUNCTION DWORD_TO_DATE2:UDINT
	VAR_INPUT
		IN :	DWORD;
	END_VAR
	DWORD_TO_DATE2 := DWORD_TO_UDINT(IN);
END_FUNCTION

PROGRAM program0
  VAR
    LocalVar0 : DWORD;
	LocalOUT  : UDINT;
  END_VAR
  	LocalOUT := DWORD_TO_DATE2(LocalVar0);
END_PROGRAM

CONFIGURATION Config0
  RESOURCE Res0 ON PLC
    TASK task0(INTERVAL := T#20ms,PRIORITY := 0);
    PROGRAM instance0 WITH task0 : program0;
  END_RESOURCE
END_CONFIGURATION

(* ---- DWORD_TO_DT.ST ---- *)
FUNCTION DWORD_TO_DT2:UDINT

	VAR_INPUT
		IN :	DWORD;
	END_VAR

	DWORD_TO_DT2 := DWORD_TO_UDINT(IN);
END_FUNCTION

PROGRAM program0
  VAR
    LocalVar0 : DWORD;
	LocalOUT  : UDINT;
  END_VAR
  	LocalOUT := DWORD_TO_DT2(LocalVar0);
END_PROGRAM

CONFIGURATION Config0
  RESOURCE Res0 ON PLC
    TASK task0(INTERVAL := T#20ms,PRIORITY := 0);
    PROGRAM instance0 WITH task0 : program0;
  END_RESOURCE
END_CONFIGURATION

(* ---- DWORD_TO_TIME.ST ---- *)
FUNCTION DWORD_TO_TIME2:TIME
	VAR_INPUT
		X :	DWORD;
	END_VAR
	DWORD_TO_TIME2 := DINT_TO_TIME(DWORD_TO_DINT(X));
END_FUNCTION

PROGRAM program0
  VAR
    LocalVar0 : DWORD;
	  LocalOUT  : TIME;
  END_VAR
  	LocalOUT := DWORD_TO_TIME2(LocalVar0);
END_PROGRAM

CONFIGURATION Config0
  RESOURCE Res0 ON PLC
    TASK task0(INTERVAL := T#20ms,PRIORITY := 0);
    PROGRAM instance0 WITH task0 : program0;
  END_RESOURCE
END_CONFIGURATION

(* ---- DWORD_TO_TOD.ST ---- *)
FUNCTION DWORD_TO_TOD2:UDINT
	VAR_INPUT
		IN :	DWORD;
	END_VAR
	DWORD_TO_TOD2 := DWORD_TO_UDINT(IN);
END_FUNCTION

PROGRAM program0
  VAR
    LocalVar0 : DWORD;
	  LocalOUT  : UDINT;
  END_VAR
  	LocalOUT := DWORD_TO_TOD2(LocalVar0);
END_PROGRAM

CONFIGURATION Config0
  RESOURCE Res0 ON PLC
    TASK task0(INTERVAL := T#20ms,PRIORITY := 0);
    PROGRAM instance0 WITH task0 : program0;
  END_RESOURCE
END_CONFIGURATION

(* ---- EASTER.ST ---- *)
FUNCTION _INT_TO_UDINT:UDINT
	VAR_INPUT
		IN :	INT;
	END_VAR

	_INT_TO_UDINT := DINT_TO_UDINT(INT_TO_DINT(IN));
END_FUNCTION

FUNCTION SET_DATE:UDINT

	VAR_INPUT
		YEAR :	INT;
		MONTH :	INT;
		DAY :	INT;
	END_VAR

	VAR
		count :	INT;
	END_VAR

	IF month > 2 THEN
		count := (month - 1) * 30;
		IF month > 7 THEN
			count := count + DWORD_TO_INT(SHR(DINT_TO_DWORD(INT_TO_DINT(month) - INT_TO_DINT(3)),1));
		ELSE
			count := count + DWORD_TO_INT(SHR(DINT_TO_DWORD(INT_TO_DINT(month) - INT_TO_DINT(4)),1));
		END_IF;
		IF SHL(INT_TO_WORD(year),14) = WORD#0 THEN
			count := count + 1;
		END_IF;
	ELSE
		count := (month - 1) * 31;
	END_IF;
	SET_DATE := (_INT_TO_UDINT(count + day - 1) + DWORD_TO_UDINT(SHR(UDINT_TO_DWORD(_INT_TO_UDINT(year) * UDINT#1461 - UDINT#2878169), 2))) * UDINT#86400;

END_FUNCTION

FUNCTION EASTER:UDINT
	VAR_INPUT
		YEAR :	INT;
	END_VAR

	VAR
		b :	INT;
		c :	INT;
		oday :	INT;
	END_VAR

	b := (204 - 11 * (year MOD 19)) MOD 30;
	IF b > 27 THEN b := b - 1; END_IF;
	c := (year + WORD_TO_INT(SHR(INT_TO_WORD(year),2)) + b - 13) MOD 7;
	oday := 28 + b - c;
	IF oday > 33 THEN
		easter := set_Date(year, 4, oday - 31);
	ELSE
		easter := set_Date(year, 3, oday);
	END_IF;
END_FUNCTION

PROGRAM program0
  VAR
    LocalVar0 : INT;
	LocalOUT  : UDINT;
  END_VAR
  	LocalOUT := EASTER(LocalVar0);
END_PROGRAM

CONFIGURATION Config0
  RESOURCE Res0 ON PLC
    TASK task0(INTERVAL := T#20ms,PRIORITY := 0);
    PROGRAM instance0 WITH task0 : program0;
  END_RESOURCE
END_CONFIGURATION

(* ---- ELLIPSE_A.ST ---- *)
FUNCTION ELLIPSE_A:REAL
	VAR_INPUT
		R1 :	REAL;
		R2 :	REAL;
	END_VAR

	ellipse_A := 3.14159265358979323846264338327950288 * R1 * R2;

END_FUNCTION

PROGRAM program0
  VAR
    LocalVar0 : REAL;
	LocalVar1 : REAL;
	  LocalOUT  : REAL;
  END_VAR
  	LocalOUT := ELLIPSE_A(LocalVar0, LocalVar1);
END_PROGRAM

CONFIGURATION Config0
  RESOURCE Res0 ON PLC
    TASK task0(INTERVAL := T#20ms,PRIORITY := 0);
    PROGRAM instance0 WITH task0 : program0;
  END_RESOURCE
END_CONFIGURATION

(* ---- ELLIPSE_C.ST ---- *)
FUNCTION ELLIPSE_C:REAL

VAR_INPUT
	R1 :	REAL;
	R2 :	REAL;
END_VAR

ELLIPSE_C := 3.14159265358979323846264338327950288 * (3.0 * (R1+R2) - SQRT((3.0 * r1 + R2) * (3.0 * r2 + r1)));

END_FUNCTION

PROGRAM program0
  VAR
    LocalVar0 : REAL;
	LocalVar1 : REAL;
	  LocalOUT  : REAL;
  END_VAR
  	LocalOUT := ELLIPSE_C(LocalVar0, LocalVar1);
END_PROGRAM

CONFIGURATION Config0
  RESOURCE Res0 ON PLC
    TASK task0(INTERVAL := T#20ms,PRIORITY := 0);
    PROGRAM instance0 WITH task0 : program0;
  END_RESOURCE
END_CONFIGURATION

(* ---- ERF.ST ---- *)
FUNCTION SGN : INT
  VAR_INPUT
    x : REAL;
  END_VAR

  IF X > 0.0 THEN
  	sgn := 1;
  ELSIF X < 0.0 THEN
  	sgn := -1;
  ELSE
  	sgn := 0;
  END_IF;
END_FUNCTION

FUNCTION ERF:REAL

	VAR_INPUT
		X :	REAL;
	END_VAR

	VAR
		x2 :	REAL;
		ax2 :	REAL;
	END_VAR

	x2 := X*X;
	ax2 := 0.147 * x2 + 1.0;
	ERF := SQRT(1.0 - EXP(-X2 * ((0.27323954473516 + aX2)/(ax2)))) * INT_TO_REAL(SGN(x));

END_FUNCTION

PROGRAM program0
  VAR
    LocalVar0 : REAL;
	  LocalOUT  : REAL;
  END_VAR
  	LocalOUT := ERF(LocalVar0);
END_PROGRAM

CONFIGURATION Config0
  RESOURCE Res0 ON PLC
    TASK task0(INTERVAL := T#20ms,PRIORITY := 0);
    PROGRAM instance0 WITH task0 : program0;
  END_RESOURCE
END_CONFIGURATION

(* ---- ERFC.ST ---- *)
FUNCTION SGN : INT
  VAR_INPUT
    x : REAL;
  END_VAR

  IF X > 0.0 THEN
  	sgn := 1;
  ELSIF X < 0.0 THEN
  	sgn := -1;
  ELSE
  	sgn := 0;
  END_IF;
END_FUNCTION

FUNCTION ERF:REAL

	VAR_INPUT
		X :	REAL;
	END_VAR

	VAR
		x2 :	REAL;
		ax2 :	REAL;
	END_VAR

	x2 := X*X;
	ax2 := 0.147 * x2 + 1.0;
	ERF := SQRT(1.0 - EXP(-X2 * ((0.27323954473516 + aX2)/(ax2)))) * INT_TO_REAL(SGN(x));

END_FUNCTION

FUNCTION ERFC:REAL
	VAR_INPUT
		X :	REAL;
	END_VAR

	ERFC := 1.0 - ERF(X);

END_FUNCTION

PROGRAM program0
  VAR
    LocalVar0 : REAL;
	  LocalOUT  : REAL;
  END_VAR
  	LocalOUT := ERFC(LocalVar0);
END_PROGRAM

CONFIGURATION Config0
  RESOURCE Res0 ON PLC
    TASK task0(INTERVAL := T#20ms,PRIORITY := 0);
    PROGRAM instance0 WITH task0 : program0;
  END_RESOURCE
END_CONFIGURATION

(* ---- EVEN.ST ---- *)
FUNCTION BIT_OF_DWORD : BOOL
  VAR_INPUT
    IN : DWORD;
    N : INT;
  END_VAR

  BIT_OF_DWORD := (SHR(in,N) AND 16#00000001) > 0;
END_FUNCTION

FUNCTION EVEN:BOOL
	VAR_INPUT
		IN :	DINT;
	END_VAR

	even := NOT BIT_OF_DWORD(DINT_TO_DWORD(in),0);
END_FUNCTION

PROGRAM program0
  VAR
    LocalVar0 : DINT;
	  LocalOUT  : BOOL;
  END_VAR
  	LocalOUT := EVEN(LocalVar0);
END_PROGRAM

CONFIGURATION Config0
  RESOURCE Res0 ON PLC
    TASK task0(INTERVAL := T#20ms,PRIORITY := 0);
    PROGRAM instance0 WITH task0 : program0;
  END_RESOURCE
END_CONFIGURATION

(* ---- EXP10.ST ---- *)
FUNCTION EXP10 : REAL
  VAR_INPUT
    x : REAL;
  END_VAR

  exp10 := EXP(X * 2.30258509299405);
  (* from OSCAT library; www.oscat.de  *)
END_FUNCTION

PROGRAM program0
  VAR
    LocalVar0 : REAL;
    CEIL5_OUT : REAL;
  END_VAR

  CEIL5_OUT := EXP10(LocalVar0);
END_PROGRAM

CONFIGURATION Config0

  RESOURCE Res0 ON PLC
    TASK task0(INTERVAL := T#20ms,PRIORITY := 0);
    PROGRAM instance0 WITH task0 : program0;
  END_RESOURCE
END_CONFIGURATION

(* ---- EXPN.ST ---- *)
FUNCTION BIT_OF_DWORD : BOOL
  VAR_INPUT
    IN : DWORD;
    N : INT;
  END_VAR

  BIT_OF_DWORD := (SHR(in,N) AND 16#00000001) > 0;
END_FUNCTION

FUNCTION EXPN:REAL

	VAR_INPUT
		X :	REAL;
		N :	INT;
	END_VAR

	VAR
		N_word :	WORD;
		X_tmp :	REAL;
		sign :	BOOL;
	END_VAR

	N_word := INT_TO_WORD(N);
	X_tmp := X;
	sign := BIT_OF_DWORD(WORD_TO_DWORD(N_word),15);
	N_word := INT_TO_WORD(ABS(N));
	IF BIT_OF_DWORD(WORD_TO_DWORD(N_word),0) THEN expn := X_tmp; ELSE expn := 1.0; END_IF;    (* N_word.X0 *)
	N_word := SHR(N_word,1);
	WHILE N_word > WORD#0 DO
		X_tmp := X_tmp * X_tmp;
		IF BIT_OF_DWORD(WORD_TO_DWORD(N_word),0) THEN expn := expn * X_tmp; END_IF;       (* N_word.X0 *)
		N_word := SHR(N_word,1);
	END_WHILE;
	IF sign THEN EXPN := 1.0 / EXPN; END_IF;

END_FUNCTION

PROGRAM program0
  VAR
    LocalVar0 : REAL;
	LocalVar1 : INT;
	LocalOUT  : REAL;
  END_VAR
  	LocalOUT := EXPN(LocalVar0, LocalVar1);
END_PROGRAM

CONFIGURATION Config0
  RESOURCE Res0 ON PLC
    TASK task0(INTERVAL := T#20ms,PRIORITY := 0);
    PROGRAM instance0 WITH task0 : program0;
  END_RESOURCE
END_CONFIGURATION

(* ---- F_LIN.ST ---- *)
FUNCTION F_LIN:REAL
	VAR_INPUT
		X :	REAL;
		A :	REAL;
		B :	REAL;
	END_VAR

	F_lin := A * X + B;
END_FUNCTION

PROGRAM program0
  VAR
    LocalVar0 : REAL;
	LocalVar1 : REAL;
	LocalVar2 : REAL;
	  LocalOUT  : REAL;
  END_VAR
  	LocalOUT := F_LIN(LocalVar0, LocalVar1, LocalVar2);
END_PROGRAM

CONFIGURATION Config0
  RESOURCE Res0 ON PLC
    TASK task0(INTERVAL := T#20ms,PRIORITY := 0);
    PROGRAM instance0 WITH task0 : program0;
  END_RESOURCE
END_CONFIGURATION

(* ---- F_LIN2.ST ---- *)
FUNCTION F_LIN2:REAL
	VAR_INPUT
		X :	REAL;
		X1 :	REAL;
		Y1 :	REAL;
		X2 :	REAL;
		Y2 :	REAL;
	END_VAR

	F_LIN2 := (Y2 - Y1) / (X2 - X1) * (X - X1) + Y1;

END_FUNCTION

PROGRAM program0
  VAR
    LocalVar0 : REAL;
	LocalVar1 : REAL;
	LocalVar2 : REAL;
	LocalVar3 : REAL;
	LocalVar4 : REAL;
	  LocalOUT  : REAL;
  END_VAR
  	LocalOUT := F_LIN2(LocalVar0, LocalVar1, LocalVar2, LocalVar3, LocalVar4);
END_PROGRAM

CONFIGURATION Config0
  RESOURCE Res0 ON PLC
    TASK task0(INTERVAL := T#20ms,PRIORITY := 0);
    PROGRAM instance0 WITH task0 : program0;
  END_RESOURCE
END_CONFIGURATION

(* ---- F_POWER.ST ---- *)
FUNCTION F_POWER:REAL
	VAR_INPUT
		A :	REAL;
		X :	REAL;
		N :	REAL;
	END_VAR

	f_power := a * EXPT(X,N);
END_FUNCTION

PROGRAM program0
  VAR
    LocalVar0 : REAL;
	LocalVar1 : REAL;
	LocalVar2 : REAL;
	  LocalOUT  : REAL;
  END_VAR
  	LocalOUT := F_POWER(LocalVar0, LocalVar1, LocalVar2);
END_PROGRAM

CONFIGURATION Config0
  RESOURCE Res0 ON PLC
    TASK task0(INTERVAL := T#20ms,PRIORITY := 0);
    PROGRAM instance0 WITH task0 : program0;
  END_RESOURCE
END_CONFIGURATION

(* ---- F_QUAD.ST ---- *)
FUNCTION F_QUAD:REAL

	VAR_INPUT
		X :	REAL;
		A :	REAL;
		B :	REAL;
		C :	REAL;
	END_VAR

	F_QUAD :=  (A * X + B) * X + C;

END_FUNCTION

PROGRAM program0
  VAR
    LocalVar0 : REAL;
	LocalVar1 : REAL;
	LocalVar2 : REAL;
	LocalVar3 : REAL;
	LocalOUT  : REAL;
  END_VAR
  	LocalOUT := F_QUAD(LocalVar0, LocalVar1, LocalVar2, LocalVar3);
END_PROGRAM

CONFIGURATION Config0
  RESOURCE Res0 ON PLC
    TASK task0(INTERVAL := T#20ms,PRIORITY := 0);
    PROGRAM instance0 WITH task0 : program0;
  END_RESOURCE
END_CONFIGURATION

(* ---- F_TO_C.ST ---- *)
FUNCTION F_TO_C:REAL
	VAR_INPUT
		FAHRENHEIT :	REAL;
	END_VAR
	F_TO_C := (fahrenheit - 32.0) * 0.5555555555555;
END_FUNCTION

PROGRAM program0
  VAR
    LocalVar0 : REAL;
	LocalOUT  : REAL;
  END_VAR
  	LocalOUT := F_TO_C(LocalVar0);
END_PROGRAM

CONFIGURATION Config0
  RESOURCE Res0 ON PLC
    TASK task0(INTERVAL := T#20ms,PRIORITY := 0);
    PROGRAM instance0 WITH task0 : program0;
  END_RESOURCE
END_CONFIGURATION

(* ---- F_TO_OM.ST ---- *)
FUNCTION F_TO_OM:REAL

	VAR_INPUT
		F :	REAL;
	END_VAR

	F_to_OM := 6.283185307179586476 * F;

END_FUNCTION

PROGRAM program0
  VAR
    LocalVar0 : REAL;
	  LocalOUT  : REAL;
  END_VAR
  	LocalOUT := F_TO_OM(LocalVar0);
END_PROGRAM

CONFIGURATION Config0
  RESOURCE Res0 ON PLC
    TASK task0(INTERVAL := T#20ms,PRIORITY := 0);
    PROGRAM instance0 WITH task0 : program0;
  END_RESOURCE
END_CONFIGURATION

(* ---- F_TO_PT.ST ---- *)
FUNCTION _REAL_TO_DWORD: DWORD
  VAR_INPUT
    X :	REAL;
  END_VAR

  IF REAL_TO_DWORD(0.5) = DWORD#1 THEN
    _REAL_TO_DWORD := REAL_TO_DWORD(x);
  ELSIF X > 0.0 THEN
    _REAL_TO_DWORD := REAL_TO_DWORD(x+0.5);
  ELSIF X < 0.0 THEN
    _REAL_TO_DWORD := REAL_TO_DWORD(x-0.5);
  ELSE
    _REAL_TO_DWORD := DWORD#0;
  END_IF;
END_FUNCTION

FUNCTION F_TO_PT:TIME
	VAR_INPUT
		F :	REAL;
	END_VAR
	F_TO_PT := DWORD_TO_TIME(_REAL_TO_DWORD(1.0 / F * 1000.0));
END_FUNCTION

PROGRAM program0
  VAR
    LocalVar0 : REAL;
	  LocalOUT  : TIME;
  END_VAR
  	LocalOUT := F_TO_PT(LocalVar0);
END_PROGRAM

CONFIGURATION Config0
  RESOURCE Res0 ON PLC
    TASK task0(INTERVAL := T#20ms,PRIORITY := 0);
    PROGRAM instance0 WITH task0 : program0;
  END_RESOURCE
END_CONFIGURATION

(* ---- FACT.ST ---- *)
FUNCTION FACT:DINT

	VAR_INPUT
		X :	INT;
	END_VAR

	CASE X OF
	00: FACT := DINT#1;
	01: FACT := DINT#1;
	02: FACT := DINT#2;
	03: FACT := DINT#6;
	04: FACT := DINT#24;
	05: FACT := DINT#120;
	06: FACT := DINT#720;
	07: FACT := DINT#5040;
	08: FACT := DINT#40320;
	09: FACT := DINT#362880;
	10: FACT := DINT#3628800;
	11: FACT := DINT#39916800;
	12: FACT := DINT#479001600;
	ELSE
		FACT := DINT#-1;
	END_CASE;

END_FUNCTION

PROGRAM program0
  VAR
    LocalVar0 : INT;
	LocalOUT  : DINT;
  END_VAR
  	LocalOUT := FACT(LocalVar0);
END_PROGRAM

CONFIGURATION Config0
  RESOURCE Res0 ON PLC
    TASK task0(INTERVAL := T#20ms,PRIORITY := 0);
    PROGRAM instance0 WITH task0 : program0;
  END_RESOURCE
END_CONFIGURATION

(* ---- FIB.ST ---- *)
FUNCTION FIB:DINT

VAR_INPUT
	X :	INT;
END_VAR

VAR
	t1 :	DINT;
	t2 :	DINT;
	X_tmp :	INT;
END_VAR

t1 := DINT#0;
t2 := DINT#0;
X_tmp := X;
IF X_tmp < 0 OR X_tmp > 46 THEN
	FIB := DINT#-1;
ELSIF X_tmp < 2 THEN
	FIB := INT_TO_DINT(X_tmp);
	RETURN;
ELSE
	t2 := DINT#1;
	WHILE X_tmp > 3 DO
		X_tmp := X_tmp - 2;
		t1 := t1 + t2;
		t2 := t1 + t2;
	END_WHILE;
	IF X_tmp > 2 THEN t1 := t1 + t2; END_IF;
	fib := t1 + t2;
END_IF;

END_FUNCTION

PROGRAM program0
  VAR
    LocalVar0 : INT;
	LocalOUT  : DINT;
  END_VAR
  	LocalOUT := FIB(LocalVar0);
END_PROGRAM

CONFIGURATION Config0
  RESOURCE Res0 ON PLC
    TASK task0(INTERVAL := T#20ms,PRIORITY := 0);
    PROGRAM instance0 WITH task0 : program0;
  END_RESOURCE
END_CONFIGURATION

(* ---- FLOOR.ST ---- *)
FUNCTION FLOOR : INT
  VAR_INPUT
    x : REAL;
  END_VAR

  FLOOR := REAL_TO_INT(X);
  IF INT_TO_REAL(FLOOR) > X THEN
  	floor := floor - 1;
  END_IF;
  (* from OSCAT library; www.oscat.de  *)
END_FUNCTION

PROGRAM program0
  VAR
    LocalVar0 : REAL;
    CEIL5_OUT : INT;
  END_VAR

  CEIL5_OUT := FLOOR(LocalVar0);
END_PROGRAM

CONFIGURATION Config0

  RESOURCE Res0 ON PLC
    TASK task0(INTERVAL := T#20ms,PRIORITY := 0);
    PROGRAM instance0 WITH task0 : program0;
  END_RESOURCE
END_CONFIGURATION

(* ---- FLOOR2.ST ---- *)
FUNCTION _REAL_TO_DINT:DINT
  VAR_INPUT
    X :	REAL;
  END_VAR

  IF REAL_TO_DINT(0.5) = DINT#1 THEN
    _REAL_TO_DINT := REAL_TO_DINT(x);
    RETURN;
  END_IF;

  IF X > 0.0 THEN
    _REAL_TO_DINT := REAL_TO_DINT(x+0.5);
  ELSIF X < 0.0 THEN
    _REAL_TO_DINT := REAL_TO_DINT(x-0.5);
  ELSE
    _REAL_TO_DINT := DINT#0;
  END_IF;
END_FUNCTION

FUNCTION FLOOR2:DINT
	VAR_INPUT
		X :	REAL;
	END_VAR

	FLOOR2 := _REAL_TO_DINT(X);
	IF DINT_TO_REAL(FLOOR2) > X THEN
		FLOOR2 := FLOOR2 - DINT#1;
	END_IF;
END_FUNCTION

PROGRAM program0
  VAR
    LocalVar0 : REAL;
    CEIL5_OUT : DINT;
  END_VAR

  CEIL5_OUT := FLOOR2(LocalVar0);
END_PROGRAM

CONFIGURATION Config0

  RESOURCE Res0 ON PLC
    TASK task0(INTERVAL := T#20ms,PRIORITY := 0);
    PROGRAM instance0 WITH task0 : program0;
  END_RESOURCE
END_CONFIGURATION

(* ---- FRACT.ST ---- *)
FUNCTION D_TRUNC : DINT
  VAR_INPUT
    x : REAL;
  END_VAR

  D_TRUNC := REAL_TO_DINT(X);
  IF X > 0.0 THEN
  	IF DINT_TO_REAL(D_TRUNC) > X THEN D_TRUNC := D_TRUNC - DINT#1; END_IF;
  ELSE
  	IF DINT_TO_REAL(D_TRUNC) < X THEN D_TRUNC := D_TRUNC + DINT#1; END_IF;
  END_IF;
END_FUNCTION

FUNCTION FRACT:REAL
	VAR_INPUT
		X :	REAL;
	END_VAR

	IF ABS(x) < 2.0E9 THEN
		FRACT := x - DINT_TO_REAL(D_TRUNC(x));
	ELSE
		FRACT := 0.0;
	END_IF;
END_FUNCTION

PROGRAM program0
  VAR
    LocalVar0 : REAL;
	LocalOUT  : REAL;
  END_VAR
  	LocalOUT := FRACT(LocalVar0);
END_PROGRAM

CONFIGURATION Config0
  RESOURCE Res0 ON PLC
    TASK task0(INTERVAL := T#20ms,PRIORITY := 0);
    PROGRAM instance0 WITH task0 : program0;
  END_RESOURCE
END_CONFIGURATION

(* ---- FRMP_B.ST ---- *)
FUNCTION FRMP_B:BYTE

	VAR_INPUT
		START :	BYTE;
		DIR :	BOOL;
		TD :	TIME;
		TR :	TIME;
	END_VAR

	IF TD < TR THEN
		FRMP_B := MIN(UDINT_TO_BYTE(DWORD_TO_UDINT(SHL(TIME_TO_DWORD(TD), 8)) / TIME_TO_UDINT(TR)), SEL(DIR, START, USINT_TO_BYTE(USINT#255 - BYTE_TO_USINT(START))));
		IF DIR THEN
			FRMP_B := USINT_TO_BYTE(BYTE_TO_USINT(START) + BYTE_TO_USINT(FRMP_B));
		ELSE
			FRMP_B := USINT_TO_BYTE(BYTE_TO_USINT(START) - BYTE_TO_USINT(FRMP_B));
		END_IF;
	ELSE
		FRMP_B := SEL(DIR, BYTE#0, BYTE#255);
	END_IF;
END_FUNCTION

PROGRAM program0
  VAR
    LocalVar0 : BYTE;
	LocalVar1 : BOOL;
	LocalVar2 : TIME;
	LocalVar3 : TIME;
    LocalOUT  : BYTE;
  END_VAR

  LocalOUT := FRMP_B(LocalVar0, LocalVar1, LocalVar2,LocalVar3);
END_PROGRAM

CONFIGURATION Config0
  RESOURCE Res0 ON PLC
    TASK task0(INTERVAL := T#20ms,PRIORITY := 0);
    PROGRAM instance0 WITH task0 : program0;
  END_RESOURCE
END_CONFIGURATION

(* ---- GAMMA.ST ---- *)
FUNCTION GAMMA:REAL
	VAR_INPUT
		X :	REAL;
	END_VAR

	IF x > 0.0 THEN
		GAMMA := SQRT(6.28318530717958647692528676655900576 / X) * EXPT(0.367879441171442 * (x + 1.0 / (12.0 * x - 0.1 / X)), X);
	END_IF;
END_FUNCTION

PROGRAM program0
  VAR
    LocalVar0 : REAL;
    LocalOUT  : REAL;
  END_VAR

  LocalOUT := GAMMA(LocalVar0);
END_PROGRAM

CONFIGURATION Config0
  RESOURCE Res0 ON PLC
    TASK task0(INTERVAL := T#20ms,PRIORITY := 0);
    PROGRAM instance0 WITH task0 : program0;
  END_RESOURCE
END_CONFIGURATION

(* ---- GAUSS.ST ---- *)
FUNCTION GAUSS:REAL

	VAR_INPUT
		X :	REAL;
		U :	REAL;
		SI :	REAL;
	END_VAR

	VAR
		temp :	REAL;
		si_inv :	REAL;
	END_VAR

	temp := X - U;
	si_inv := 1.0  / si;
	GAUSS := EXP(Temp * Temp * si_inv * SI_inv * - 0.5) * 0.39894228 * si_inv;

END_FUNCTION

PROGRAM program0
  VAR
    X :	REAL;
	U :	REAL;
	SI :	REAL;
    LocalOUT  : REAL;
  END_VAR

  LocalOUT := GAUSS(X, U, SI);
END_PROGRAM

CONFIGURATION Config0
  RESOURCE Res0 ON PLC
    TASK task0(INTERVAL := T#20ms,PRIORITY := 0);
    PROGRAM instance0 WITH task0 : program0;
  END_RESOURCE
END_CONFIGURATION

(* ---- GAUSSCD.ST ---- *)
FUNCTION SGN : INT
  VAR_INPUT
    x : REAL;
  END_VAR

  IF X > 0.0 THEN
  	sgn := 1;
  ELSIF X < 0.0 THEN
  	sgn := -1;
  ELSE
  	sgn := 0;
  END_IF;
END_FUNCTION

FUNCTION ERF:REAL

	VAR_INPUT
		X :	REAL;
	END_VAR

	VAR
		x2 :	REAL;
		ax2 :	REAL;
	END_VAR

	x2 := X*X;
	ax2 := 0.147 * x2 + 1.0;
	ERF := SQRT(1.0 - EXP(-X2 * ((0.27323954473516 + aX2)/(ax2)))) * INT_TO_REAL(SGN(x));

END_FUNCTION

FUNCTION GAUSSCD:REAL

	VAR_INPUT
		X :	REAL;
		U :	REAL;
		SI :	REAL;
	END_VAR

	GAUSSCD := (ERF((X - U) / (SI * 1.414213562)) + 1.0) * 0.5;

END_FUNCTION

PROGRAM program0
  VAR
    X :	REAL;
	U :	REAL;
	SI :	REAL;
    LocalOUT  : REAL;
  END_VAR

  LocalOUT := GAUSSCD(X, U, SI);
END_PROGRAM

CONFIGURATION Config0
  RESOURCE Res0 ON PLC
    TASK task0(INTERVAL := T#20ms,PRIORITY := 0);
    PROGRAM instance0 WITH task0 : program0;
  END_RESOURCE
END_CONFIGURATION

(* ---- GCD.ST ---- *)
FUNCTION GCD:INT

	VAR_INPUT
		A :	DINT;
		B :	DINT;
	END_VAR

	VAR
		t :	DINT;
		_A :	DINT;
		_B :	DINT;
	END_VAR

	_A := A;
	_B := B;

	IF _A = DINT#0 THEN
		GCD := DINT_TO_INT(ABS(_B));
	ELSIF _B = DINT#0 THEN
		GCD := DINT_TO_INT(ABS(_A));
	ELSE
		_A := ABS(_A);
		_B := ABS(_B);
		GCD := 1;

		WHILE NOT((DINT_TO_DWORD(_A) AND DWORD#1) > DWORD#0 OR (DINT_TO_DWORD(_B) AND DWORD#1) > DWORD#0) DO
			_A := DWORD_TO_DINT(SHR(DINT_TO_DWORD(_A),1));
			_B := DWORD_TO_DINT(SHR(DINT_TO_DWORD(_B),1));
			GCD := DWORD_TO_INT(SHR(INT_TO_DWORD(GCD),1));
		END_WHILE;
		WHILE _A > DINT#0 DO
			IF NOT((DINT_TO_DWORD(_A) AND DWORD#1) > DWORD#0) THEN
				_A := DWORD_TO_DINT(SHR(DINT_TO_DWORD(_A),1));
			ELSIF NOT((DINT_TO_DWORD(_B) AND DWORD#1) > DWORD#0) THEN
				_B := DWORD_TO_DINT(SHR(DINT_TO_DWORD(_B),1));
			ELSE
				t := DWORD_TO_DINT(SHR(DINT_TO_DWORD(ABS(_A-_B)),1));
				IF _A < _B THEN
					_B := t;
				ELSE
					_A := t;
				END_IF;
			END_IF;
		END_WHILE;
		GCD := GCD * DINT_TO_INT(_B);
	END_IF;

END_FUNCTION

PROGRAM program0
  VAR
    A :	DINT;
	B :	DINT;
    LocalOUT  : INT;
  END_VAR

  LocalOUT := GCD(A, B);
END_PROGRAM

CONFIGURATION Config0
  RESOURCE Res0 ON PLC
    TASK task0(INTERVAL := T#20ms,PRIORITY := 0);
    PROGRAM instance0 WITH task0 : program0;
  END_RESOURCE
END_CONFIGURATION

(* ---- GDF.ST ---- *)
FUNCTION GDF:REAL

	VAR_INPUT
		X :	REAL;
	END_VAR

	IF X = 0.0 THEN
		GDF := 0.0;
	ELSIF X > 15.0 THEN
		GDF := 1.5707963267949;
	ELSIF X < -15.0 THEN
		GDF := -1.5707963267949;
	ELSE
		GDF := ATAN(EXP(X)) * 2.0 - 1.5707963267949;
	END_IF;

END_FUNCTION

PROGRAM program0
  VAR
    X :	REAL;
    LocalOUT  : REAL;
  END_VAR

  LocalOUT := GDF(X);
END_PROGRAM

CONFIGURATION Config0
  RESOURCE Res0 ON PLC
    TASK task0(INTERVAL := T#20ms,PRIORITY := 0);
    PROGRAM instance0 WITH task0 : program0;
  END_RESOURCE
END_CONFIGURATION

(* ---- GEO_TO_DEG.ST ---- *)
FUNCTION GEO_TO_DEG:REAL

	VAR_INPUT
		D :	INT;
		M :	INT;
		SEC :	REAL;
	END_VAR

	GEO_TO_DEG := INT_TO_REAL(D) + INT_TO_REAL(M) * 0.016666666666667 + sec * 0.00027777777777778;

END_FUNCTION

PROGRAM program0
  VAR
    D :	INT;
	M :	INT;
	SEC :	REAL;
    LocalOUT  : REAL;
  END_VAR

  LocalOUT := GEO_TO_DEG(D, M, SEC);
END_PROGRAM

CONFIGURATION Config0
  RESOURCE Res0 ON PLC
    TASK task0(INTERVAL := T#20ms,PRIORITY := 0);
    PROGRAM instance0 WITH task0 : program0;
  END_RESOURCE
END_CONFIGURATION

(* ---- GOLD.ST ---- *)
FUNCTION GOLD:REAL

	VAR_INPUT
		X :	REAL;
	END_VAR

	GOLD := (X + SQRT(X*X + 4.0)) * 0.5;

END_FUNCTION

PROGRAM program0
  VAR
   	X :	REAL;
    LocalOUT  : REAL;
  END_VAR

  LocalOUT := GOLD(X);
END_PROGRAM

CONFIGURATION Config0
  RESOURCE Res0 ON PLC
    TASK task0(INTERVAL := T#20ms,PRIORITY := 0);
    PROGRAM instance0 WITH task0 : program0;
  END_RESOURCE
END_CONFIGURATION

(* ---- GRAY_TO_BYTE.ST ---- *)
FUNCTION GRAY_TO_BYTE:BYTE

	VAR_INPUT
		IN :	BYTE;
	END_VAR

	GRAY_TO_BYTE := SHR(IN,4) XOR IN;
	GRAY_TO_BYTE := SHR(GRAY_TO_BYTE,2) XOR GRAY_TO_BYTE;
	GRAY_TO_BYTE := SHR(GRAY_TO_BYTE,1) XOR GRAY_TO_BYTE;

END_FUNCTION

PROGRAM program0
  VAR
   	IN :	BYTE;
    LocalOUT  : BYTE;
  END_VAR

  LocalOUT := GRAY_TO_BYTE(IN);
END_PROGRAM

CONFIGURATION Config0
  RESOURCE Res0 ON PLC
    TASK task0(INTERVAL := T#20ms,PRIORITY := 0);
    PROGRAM instance0 WITH task0 : program0;
  END_RESOURCE
END_CONFIGURATION

(* ---- HEAT_INDEX.ST ---- *)
FUNCTION C_TO_F:REAL
	VAR_INPUT
		CELSIUS :	REAL;
	END_VAR

	C_TO_F := celsius * 1.8 + 32.0;
END_FUNCTION

FUNCTION F_TO_C:REAL
	VAR_INPUT
		FAHRENHEIT :	REAL;
	END_VAR
	F_TO_C := (fahrenheit - 32.0) * 0.5555555555555;
END_FUNCTION

FUNCTION HEAT_INDEX:REAL

	VAR_INPUT
		T :	REAL;
		RH :	REAL;
	END_VAR

	VAR
		RH2 :	REAL;
		T2 :	REAL;
		TX :	REAL;
	END_VAR

	IF RH < 20.0 OR T < 20.0 THEN
		HEAT_INDEX := T;
	ELSE
		TX := T;
		RH2 := RH * RH;
		TX := C_TO_F(TX);
		T2 := TX * TX;
		HEAT_INDEX := -42.379 + 2.04901523 * TX - 6.83783E-3 * T2
				+ RH * (10.1433127 - 0.22475541 * TX + 1.22874E-3 * T2)
				+ RH2 * (8.5282E-4 * TX - 5.481717E-2 - 1.99E-6 * T2);
		HEAT_INDEX := F_TO_C(HEAT_INDEX);
	END_IF;

END_FUNCTION

PROGRAM program0
  VAR
    T :	REAL;
	RH :	REAL;
    CEIL5_OUT : REAL;
  END_VAR

  CEIL5_OUT := HEAT_INDEX(T, RH);
END_PROGRAM

CONFIGURATION Config0

  RESOURCE Res0 ON PLC
    TASK task0(INTERVAL := T#20ms,PRIORITY := 0);
    PROGRAM instance0 WITH task0 : program0;
  END_RESOURCE
END_CONFIGURATION

(* ---- HOUR.ST ---- *)
FUNCTION HOUR:INT
	VAR_INPUT
		ITOD :	UDINT;
	END_VAR
	hour := UDINT_TO_INT(itod / UDINT#3600000);
END_FUNCTION

PROGRAM program0
  VAR
	  ITOD :	UDINT;
    CEIL5_OUT : INT;
  END_VAR

  CEIL5_OUT := HOUR(ITOD);
END_PROGRAM

CONFIGURATION Config0

  RESOURCE Res0 ON PLC
    TASK task0(INTERVAL := T#20ms,PRIORITY := 0);
    PROGRAM instance0 WITH task0 : program0;
  END_RESOURCE
END_CONFIGURATION

(* ---- HOUR_OF_DT.ST ---- *)
FUNCTION HOUR_OF_DT:INT
	VAR_INPUT
		XDT :	UDINT;
	END_VAR

	HOUR_OF_DT := UDINT_TO_INT((XDT MOD UDINT#86400) / UDINT#3600);
END_FUNCTION

PROGRAM program0
  VAR
    LocalVar0 : UDINT;
	LocalOUT  : INT;
  END_VAR
  	LocalOUT := HOUR_OF_DT(LocalVar0);
END_PROGRAM

CONFIGURATION Config0
  RESOURCE Res0 ON PLC
    TASK task0(INTERVAL := T#20ms,PRIORITY := 0);
    PROGRAM instance0 WITH task0 : program0;
  END_RESOURCE
END_CONFIGURATION

(* ---- HOUR_TO_TIME.ST ---- *)
FUNCTION _REAL_TO_UDINT:UDINT
	VAR_INPUT
		X :	REAL;
	END_VAR

	IF REAL_TO_UDINT(0.5) = UDINT#1 THEN
		_REAL_TO_UDINT := REAL_TO_UDINT(x);
	ELSIF X > 0.0 THEN
		_REAL_TO_UDINT := REAL_TO_UDINT(x+0.5);
	ELSIF X < 0.0 THEN
		_REAL_TO_UDINT := REAL_TO_UDINT(x-0.5);
	ELSE
		_REAL_TO_UDINT := UDINT#0;
  	END_IF;
END_FUNCTION

FUNCTION HOUR_TO_TIME:TIME

	VAR_INPUT
		IN :	REAL;
	END_VAR

	hour_to_time := UDINT_TO_TIME(_REAL_TO_UDINT(IN * 3600000.0));

END_FUNCTION

PROGRAM program0

	VAR
		IN :	REAL;
		CEIL5_OUT : TIME;
	END_VAR

  	CEIL5_OUT := HOUR_TO_TIME(IN);

END_PROGRAM

CONFIGURATION Config0

	RESOURCE Res0 ON PLC
		TASK task0(INTERVAL := T#20ms,PRIORITY := 0);
		PROGRAM instance0 WITH task0 : program0;
	END_RESOURCE

END_CONFIGURATION

(* ---- HOUR_TO_TOD.ST ---- *)
FUNCTION _REAL_TO_UDINT:UDINT
	VAR_INPUT
		X :	REAL;
	END_VAR

	IF REAL_TO_UDINT(0.5) = UDINT#1 THEN
		_REAL_TO_UDINT := REAL_TO_UDINT(x);
	ELSIF X > 0.0 THEN
		_REAL_TO_UDINT := REAL_TO_UDINT(x+0.5);
	ELSIF X < 0.0 THEN
		_REAL_TO_UDINT := REAL_TO_UDINT(x-0.5);
	ELSE
		_REAL_TO_UDINT := UDINT#0;
	END_IF;

END_FUNCTION

FUNCTION HOUR_TO_TOD:UDINT

	VAR_INPUT
		IN :	REAL;
	END_VAR

	hour_to_tod := _REAL_TO_UDINT(IN * 3600000.00);

END_FUNCTION

PROGRAM program0
	VAR
		IN :	REAL;
		CEIL5_OUT : UDINT;
	END_VAR

  	CEIL5_OUT := HOUR_TO_TOD(IN);
END_PROGRAM

CONFIGURATION Config0

  RESOURCE Res0 ON PLC
    TASK task0(INTERVAL := T#20ms,PRIORITY := 0);
    PROGRAM instance0 WITH task0 : program0;
  END_RESOURCE

END_CONFIGURATION

(* ---- HYPOT.ST ---- *)
FUNCTION HYPOT:REAL
	VAR_INPUT
		X :	REAL;
		Y :	REAL;
	END_VAR

	HYPOT := SQRT(x*x + y*y);
END_FUNCTION

PROGRAM program0
  VAR
    LocalVar0 : REAL;
    LocalVar1 : REAL;
    CEIL5_OUT : REAL;
  END_VAR

  CEIL5_OUT := HYPOT(LocalVar0, LocalVar1);
END_PROGRAM

CONFIGURATION Config0

  RESOURCE Res0 ON PLC
    TASK task0(INTERVAL := T#20ms,PRIORITY := 0);
    PROGRAM instance0 WITH task0 : program0;
  END_RESOURCE
END_CONFIGURATION

(* ---- INC.ST ---- *)
FUNCTION INC:INT
	VAR_INPUT
		X :	INT;
		D :	INT;
		M :	INT;
	END_VAR

	inc := (X + D + M + 1) MOD (M + 1);
END_FUNCTION

PROGRAM program0
  VAR
    LocalVar0 : INT;
	LocalVar1 : INT;
	LocalVar2 : INT;
	LocalOUT  : INT;
  END_VAR
  	LocalOUT := INC(LocalVar0, LocalVar1,LocalVar2);
END_PROGRAM

CONFIGURATION Config0
  RESOURCE Res0 ON PLC
    TASK task0(INTERVAL := T#20ms,PRIORITY := 0);
    PROGRAM instance0 WITH task0 : program0;
  END_RESOURCE
END_CONFIGURATION

(* ---- INC1.ST ---- *)
FUNCTION INC1:INT

	VAR_INPUT
		X :	INT;
		N :	INT;
	END_VAR

	IF X >= N - 1 THEN
		INC1 := 0;
	ELSE
		INC1 := X + 1;
	END_IF;
END_FUNCTION

PROGRAM program0
  VAR
	X :	INT;
	N :	INT;
    CEIL5_OUT : INT;
  END_VAR

  CEIL5_OUT := INC1(X, N);
END_PROGRAM

CONFIGURATION Config0

  RESOURCE Res0 ON PLC
    TASK task0(INTERVAL := T#20ms,PRIORITY := 0);
    PROGRAM instance0 WITH task0 : program0;
  END_RESOURCE
END_CONFIGURATION

(* ---- INC2.ST ---- *)
FUNCTION INC2:INT

	VAR_INPUT
		X :	INT;
		D :	INT;
		L :	INT;
		U :	INT;
	END_VAR

	VAR
		tmp :	INT;
	END_VAR

	tmp := U - L + 1;
	INC2 := (X + D - L + tmp) MOD tmp + L;

END_FUNCTION

PROGRAM program0
	VAR
		X :	INT;
		D :	INT;
		L :	INT;
		U :	INT;
		CEIL5_OUT : INT;
	END_VAR

  	CEIL5_OUT := INC2(X, D, L, U);
END_PROGRAM

CONFIGURATION Config0

	RESOURCE Res0 ON PLC
		TASK task0(INTERVAL := T#20ms,PRIORITY := 0);
		PROGRAM instance0 WITH task0 : program0;
	END_RESOURCE

END_CONFIGURATION

(* ---- INT_TO_BCDC.ST ---- *)
FUNCTION INT_TO_BCDC:BYTE

	VAR_INPUT
		IN :	INT;
	END_VAR

	INT_TO_BCDC := SHL(INT_TO_BYTE(IN / INT#10),4) OR INT_TO_BYTE(in MOD INT#10);

END_FUNCTION

PROGRAM program0

	VAR
		IN :	INT;
		OUT : BYTE;
	END_VAR

	OUT := INT_TO_BCDC(IN);

END_PROGRAM

CONFIGURATION Config0

	RESOURCE Res0 ON PLC
		TASK task0(INTERVAL := T#20ms,PRIORITY := 0);
		PROGRAM instance0 WITH task0 : program0;
	END_RESOURCE

END_CONFIGURATION

(* ---- INT_TO_TIME.ST ---- *)
FUNCTION _INT_TO_TIME:TIME

	VAR_INPUT
		IN :	INT;
	END_VAR

	_INT_TO_TIME := DINT_TO_TIME(INT_TO_DINT(IN));

END_FUNCTION

PROGRAM program0
	VAR
		IN :	INT;
		OUT : TIME;
	END_VAR

	OUT := _INT_TO_TIME(IN);
END_PROGRAM

CONFIGURATION Config0

	RESOURCE Res0 ON PLC
		TASK task0(INTERVAL := T#20ms,PRIORITY := 0);
		PROGRAM instance0 WITH task0 : program0;
	END_RESOURCE

END_CONFIGURATION

(* ---- INV.ST ---- *)
FUNCTION INV:REAL

	VAR_INPUT
		X :	REAL;
	END_VAR

	IF X <> 0.0 THEN INV := 1.0 / X; END_IF;

END_FUNCTION

PROGRAM program0
	VAR
		X :	REAL;
		OUT : REAL;
	END_VAR

	OUT := INV(X);
END_PROGRAM

CONFIGURATION Config0

	RESOURCE Res0 ON PLC
		TASK task0(INTERVAL := T#20ms,PRIORITY := 0);
		PROGRAM instance0 WITH task0 : program0;
	END_RESOURCE

END_CONFIGURATION

(* ---- IP4_CHECK.ST ---- *)
FUNCTION IP4_CHECK:BOOL

	VAR_INPUT
		NIP :	DWORD;
		LIP :	DWORD;
		SM :	DWORD;
	END_VAR

	IP4_CHECK := (NIP AND sm) = (LIP AND SM);

END_FUNCTION

PROGRAM program0
	VAR
		NIP :	DWORD;
		LIP :	DWORD;
		SM :	DWORD;
		CEIL5_OUT : BOOL;
	END_VAR

  	CEIL5_OUT := IP4_CHECK(NIP, LIP, SM);
END_PROGRAM

CONFIGURATION Config0

  RESOURCE Res0 ON PLC
    TASK task0(INTERVAL := T#20ms,PRIORITY := 0);
    PROGRAM instance0 WITH task0 : program0;
  END_RESOURCE
END_CONFIGURATION

(* ---- IS_URLCHR.ST ---- *)
FUNCTION IS_URLCHR:BOOL

	VAR_INPUT
		IN :	BYTE;
	END_VAR

	IS_URLCHR := ((IN>BYTE#47) AND (IN<BYTE#58)) OR ((IN>BYTE#64) AND (IN<BYTE#91)) OR ((IN>BYTE#96) AND (IN<BYTE#123)) OR (in=BYTE#126) OR (in=BYTE#95) OR (in=BYTE#45) OR (in=BYTE#46);

END_FUNCTION

PROGRAM program0
	VAR
		IN :	BYTE;
		CEIL5_OUT : BOOL;
	END_VAR

  	CEIL5_OUT := IS_URLCHR(IN);
END_PROGRAM

CONFIGURATION Config0

  RESOURCE Res0 ON PLC
    TASK task0(INTERVAL := T#20ms,PRIORITY := 0);
    PROGRAM instance0 WITH task0 : program0;
  END_RESOURCE
END_CONFIGURATION

(* ---- ISC_ALPHA.ST ---- *)
FUNCTION SETUP_EXTENDED_ASCII:BOOL

	VAR_INPUT
		X :	BOOL;
	END_VAR

	SETUP_EXTENDED_ASCII := X OR TRUE;

END_FUNCTION

FUNCTION ISC_ALPHA:BOOL

	VAR_INPUT
		IN :	BYTE;
	END_VAR

	IF SETUP_EXTENDED_ASCII(FALSE) THEN
		ISC_ALPHA := (in > BYTE#64 AND in < BYTE#91) OR (in > BYTE#191  AND in <> BYTE#215 AND in <> BYTE#247) OR (in > BYTE#96 AND in < BYTE#123);
	ELSE
		ISC_ALPHA := (IN > BYTE#64 AND IN < BYTE#91) OR (in > BYTE#96 AND in < BYTE#123);
	END_IF;

END_FUNCTION

PROGRAM program0
	VAR
		IN : BYTE;
		OUT : BOOL;
	END_VAR

	OUT := ISC_ALPHA(IN);
END_PROGRAM

CONFIGURATION Config0

	RESOURCE Res0 ON PLC
		TASK task0(INTERVAL := T#20ms,PRIORITY := 0);
		PROGRAM instance0 WITH task0 : program0;
	END_RESOURCE

END_CONFIGURATION

(* ---- ISC_CTRL.ST ---- *)
FUNCTION ISC_CTRL:BOOL

	VAR_INPUT
		IN :	BYTE;
	END_VAR

	ISC_CTRL := IN < BYTE#32 OR IN = BYTE#127;

END_FUNCTION

PROGRAM program0
	VAR
		IN : BYTE;
		OUT : BOOL;
	END_VAR

	OUT := ISC_CTRL(IN);
END_PROGRAM

CONFIGURATION Config0

	RESOURCE Res0 ON PLC
		TASK task0(INTERVAL := T#20ms,PRIORITY := 0);
		PROGRAM instance0 WITH task0 : program0;
	END_RESOURCE

END_CONFIGURATION

(* ---- ISC_HEX.ST ---- *)
FUNCTION ISC_HEX:BOOL

	VAR_INPUT
		IN :	BYTE;
	END_VAR

	ISC_HEX := (IN > BYTE#47 AND IN < BYTE#58) OR (IN > BYTE#64 AND IN < BYTE#71) OR (IN > BYTE#96 AND IN < BYTE#103);

END_FUNCTION

PROGRAM program0
	VAR
		IN : BYTE;
		OUT : BOOL;
	END_VAR

	OUT := ISC_HEX(IN);
END_PROGRAM

CONFIGURATION Config0

	RESOURCE Res0 ON PLC
		TASK task0(INTERVAL := T#20ms,PRIORITY := 0);
		PROGRAM instance0 WITH task0 : program0;
	END_RESOURCE

END_CONFIGURATION

(* ---- ISC_LOWER.ST ---- *)
FUNCTION SETUP_EXTENDED_ASCII:BOOL

	VAR_INPUT
		X :	BOOL;
	END_VAR

	SETUP_EXTENDED_ASCII := X OR TRUE;

END_FUNCTION

FUNCTION ISC_LOWER:BOOL

	VAR_INPUT
		IN :	BYTE;
	END_VAR

	IF SETUP_EXTENDED_ASCII(FALSE) THEN
		ISC_LOWER := ((in > BYTE#96) AND (in < BYTE#123)) OR ((in > BYTE#222) AND (in <> BYTE#247));
	ELSE
		ISC_LOWER := ((in > BYTE#96) AND (in < BYTE#123));
	END_IF;

END_FUNCTION

PROGRAM program0
	VAR
		IN : BYTE;
		OUT : BOOL;
	END_VAR

	OUT := ISC_LOWER(IN);
END_PROGRAM

CONFIGURATION Config0

	RESOURCE Res0 ON PLC
		TASK task0(INTERVAL := T#20ms,PRIORITY := 0);
		PROGRAM instance0 WITH task0 : program0;
	END_RESOURCE

END_CONFIGURATION

(* ---- ISC_NUM.ST ---- *)
FUNCTION ISC_NUM:BOOL

	VAR_INPUT
		IN :	BYTE;
	END_VAR

	ISC_NUM := IN > BYTE#47 AND IN < BYTE#58;

END_FUNCTION

PROGRAM program0
	VAR
		IN : BYTE;
		OUT : BOOL;
	END_VAR

	OUT := ISC_NUM(IN);
END_PROGRAM

CONFIGURATION Config0

	RESOURCE Res0 ON PLC
		TASK task0(INTERVAL := T#20ms,PRIORITY := 0);
		PROGRAM instance0 WITH task0 : program0;
	END_RESOURCE

END_CONFIGURATION

(* ---- ISC_UPPER.ST ---- *)
FUNCTION SETUP_EXTENDED_ASCII:BOOL

	VAR_INPUT
		X :	BOOL;
	END_VAR

	SETUP_EXTENDED_ASCII := X OR TRUE;

END_FUNCTION

FUNCTION ISC_UPPER:BOOL

	VAR_INPUT
		IN :	BYTE;
	END_VAR

	IF SETUP_EXTENDED_ASCII(FALSE) THEN
		ISC_UPPER :=  ((in > BYTE#64) AND (in < BYTE#91)) OR (((in > BYTE#191) AND (in < BYTE#223)) AND (in <> BYTE#215));
	ELSE
		ISC_UPPER := ((in > BYTE#64) AND (in < BYTE#91));
	END_IF;

END_FUNCTION

PROGRAM program0
	VAR
		IN : BYTE;
		OUT : BOOL;
	END_VAR

	OUT := ISC_UPPER(IN);
END_PROGRAM

CONFIGURATION Config0

	RESOURCE Res0 ON PLC
		TASK task0(INTERVAL := T#20ms,PRIORITY := 0);
		PROGRAM instance0 WITH task0 : program0;
	END_RESOURCE

END_CONFIGURATION

(* ---- JD2000.ST ---- *)
FUNCTION JD2000:REAL

	VAR_INPUT
		DTI :	UDINT;
	END_VAR

	JD2000 := UDINT_TO_REAL(DTI - UDINT#946728000) / 86400.0;

END_FUNCTION

PROGRAM program0
	VAR
		DTI :	UDINT;
		OUT : REAL;
	END_VAR

	OUT := JD2000(DTI);
END_PROGRAM

CONFIGURATION Config0

	RESOURCE Res0 ON PLC
		TASK task0(INTERVAL := T#20ms,PRIORITY := 0);
		PROGRAM instance0 WITH task0 : program0;
	END_RESOURCE

END_CONFIGURATION

(* ---- K_TO_C.ST ---- *)
FUNCTION K_TO_C:REAL

	VAR_INPUT
		KELVIN :	REAL;
	END_VAR

	K_to_C := Kelvin + 273.15;

END_FUNCTION

PROGRAM program0
	VAR
		KELVIN : REAL;
		OUT : REAL;
	END_VAR

	OUT := K_TO_C(KELVIN);
END_PROGRAM

CONFIGURATION Config0

	RESOURCE Res0 ON PLC
		TASK task0(INTERVAL := T#20ms,PRIORITY := 0);
		PROGRAM instance0 WITH task0 : program0;
	END_RESOURCE

END_CONFIGURATION

(* ---- KMH_TO_MS.ST ---- *)
FUNCTION KMH_TO_MS:REAL

	VAR_INPUT
		KMH :	REAL;
	END_VAR

	KMH_TO_MS := kmh * 0.2777777777777;

END_FUNCTION

PROGRAM program0
	VAR
		KMH : REAL;
		OUT : REAL;
	END_VAR

	OUT := KMH_TO_MS(KMH);
END_PROGRAM

CONFIGURATION Config0

	RESOURCE Res0 ON PLC
		TASK task0(INTERVAL := T#20ms,PRIORITY := 0);
		PROGRAM instance0 WITH task0 : program0;
	END_RESOURCE

END_CONFIGURATION

(* ---- LANGEVIN.ST ---- *)
FUNCTION COTH:REAL

	VAR_INPUT
		X :	REAL;
	END_VAR

	IF X > 20.0 THEN
		COTH :=1.0;
	ELSIF X < -20.0 THEN
		COTH := -1.0;
	ELSE
		COTH := 1.0 + 2.0 / (EXP(X * 2.0) - 1.0);
	END_IF;

END_FUNCTION

FUNCTION LANGEVIN:REAL

	VAR_INPUT
		X :	REAL;
	END_VAR

	IF X = 0.0 THEN
		LANGEVIN := 0.0;
	ELSE
		LANGEVIN := COTH(X) - 1.0 / X;
	END_IF;

END_FUNCTION

PROGRAM program0
	VAR
		X :	REAL;
		OUT : REAL;
	END_VAR

	OUT := LANGEVIN(X);
END_PROGRAM

CONFIGURATION Config0

	RESOURCE Res0 ON PLC
		TASK task0(INTERVAL := T#20ms,PRIORITY := 0);
		PROGRAM instance0 WITH task0 : program0;
	END_RESOURCE

END_CONFIGURATION

(* ---- LEAP_DAY.ST ---- *)
FUNCTION LEAP_DAY:BOOL

	VAR_INPUT
		IDATE :	UDINT;
	END_VAR

	LEAP_DAY := IDATE MOD UDINT#126230400 = UDINT#68169600;

END_FUNCTION

PROGRAM program0
	VAR
		IDATE :	UDINT;
		OUT : BOOL;
	END_VAR

	OUT := LEAP_DAY(IDATE);
END_PROGRAM

CONFIGURATION Config0

	RESOURCE Res0 ON PLC
		TASK task0(INTERVAL := T#20ms,PRIORITY := 0);
		PROGRAM instance0 WITH task0 : program0;
	END_RESOURCE

END_CONFIGURATION

(* ---- LEAP_OF_DATE.ST ---- *)
FUNCTION LEAP_OF_DATE:BOOL

	VAR_INPUT
		IDATE :	UDINT;
	END_VAR

	LEAP_OF_DATE := SHL(UDINT_TO_DWORD((idate + UDINT#43200) / UDINT#31557600), 30) = DWORD#16#80000000;

END_FUNCTION

PROGRAM program0
  VAR
    LocalVar0 : UDINT;
	LocalOUT  : BOOL;
  END_VAR
  	LocalOUT := LEAP_OF_DATE(LocalVar0);
END_PROGRAM

CONFIGURATION Config0
  RESOURCE Res0 ON PLC
    TASK task0(INTERVAL := T#20ms,PRIORITY := 0);
    PROGRAM instance0 WITH task0 : program0;
  END_RESOURCE
END_CONFIGURATION

(* ---- LEAP_YEAR.ST ---- *)
FUNCTION LEAP_YEAR:BOOL

  VAR_INPUT
    YEAR :	INT;
  END_VAR

  IF (year MOD INT#400) = INT#00 THEN
    leap_year := TRUE;
  ELSIF (year MOD INT#100) = INT#00 THEN
    leap_year := FALSE;
  ELSIF (year MOD INT#04) = INT#00 THEN
    leap_year := TRUE;
  ELSE
    leap_year := FALSE;
  END_IF;

END_FUNCTION

PROGRAM program0
	VAR
		YEAR :	INT;
		OUT : BOOL;
	END_VAR

	OUT := LEAP_YEAR(YEAR);
END_PROGRAM

CONFIGURATION Config0

	RESOURCE Res0 ON PLC
		TASK task0(INTERVAL := T#20ms,PRIORITY := 0);
		PROGRAM instance0 WITH task0 : program0;
	END_RESOURCE

END_CONFIGURATION

(* ---- LTIME_TO_UTC.ST ---- *)
FUNCTION _INT_TO_UDINT:UDINT
	VAR_INPUT
		IN :	INT;
	END_VAR

	_INT_TO_UDINT := DINT_TO_UDINT(INT_TO_DINT(IN));
END_FUNCTION

FUNCTION LTIME_TO_UTC:UDINT

	VAR_INPUT
		LTIME :	UDINT;
		DST :	BOOL;
		TIME_ZONE_OFFSET :	INT;
	END_VAR

	LTIME_TO_UTC := LTIME - _INT_TO_UDINT(TIME_ZONE_OFFSET * 60);
	IF DST THEN LTIME_TO_UTC := LTIME_TO_UTC - UDINT#3600; END_IF;

END_FUNCTION

PROGRAM program0
	VAR
		LTIME :	UDINT;
		DST :	BOOL;
		TIME_ZONE_OFFSET :	INT;
		CEIL5_OUT : UDINT;
	END_VAR

  CEIL5_OUT := LTIME_TO_UTC(LTIME, DST, TIME_ZONE_OFFSET);
END_PROGRAM

CONFIGURATION Config0

  RESOURCE Res0 ON PLC
    TASK task0(INTERVAL := T#20ms,PRIORITY := 0);
    PROGRAM instance0 WITH task0 : program0;
  END_RESOURCE
END_CONFIGURATION

(* ---- MANUAL.ST ---- *)
FUNCTION MANUAL:BOOL

	VAR_INPUT
		_IN :	BOOL;
		_ON :	BOOL;
		OFF :	BOOL;
	END_VAR

	MANUAL := NOT OFF AND (_IN OR _ON);

END_FUNCTION

PROGRAM program0
	VAR
		_IN :	BOOL;
		_ON :	BOOL;
		OFF :	BOOL;

		OUT : BOOL;
	END_VAR

	OUT := MANUAL(_IN, _ON, OFF);

END_PROGRAM

CONFIGURATION Config0

	RESOURCE Res0 ON PLC
		TASK task0(INTERVAL := T#20ms,PRIORITY := 0);
		PROGRAM instance0 WITH task0 : program0;
	END_RESOURCE

END_CONFIGURATION

(* ---- MAX3.ST ---- *)
FUNCTION MAX3:REAL

	VAR_INPUT
		IN1 :	REAL;
		IN2 :	REAL;
		IN3 :	REAL;
	END_VAR

	MAX3 := MAX(MAX(IN1,IN2),IN3);

END_FUNCTION

PROGRAM program0
	VAR
		IN1 :	REAL;
		IN2 :	REAL;
		IN3 :	REAL;

		OUT : REAL;
	END_VAR

	OUT := MAX3(IN1, IN2, IN3);

END_PROGRAM

CONFIGURATION Config0

	RESOURCE Res0 ON PLC
		TASK task0(INTERVAL := T#20ms,PRIORITY := 0);
		PROGRAM instance0 WITH task0 : program0;
	END_RESOURCE

END_CONFIGURATION

(* ---- MAX_TIME.ST ---- *)
FUNCTION _MAX_TIME:TIME

	VAR_INPUT
		IN1 :	TIME;
		IN2 :	TIME;
	END_VAR

	_MAX_TIME := SEL_TIME(IN1 < IN2,IN1,IN2);

END_FUNCTION

PROGRAM program0
	VAR
		IN1 :	TIME;
		IN2 :	TIME;

		OUT : TIME;
	END_VAR

	OUT := _MAX_TIME(IN1, IN2);

END_PROGRAM

CONFIGURATION Config0

	RESOURCE Res0 ON PLC
		TASK task0(INTERVAL := T#20ms,PRIORITY := 0);
		PROGRAM instance0 WITH task0 : program0;
	END_RESOURCE

END_CONFIGURATION

(* ---- MID3.ST ---- *)
FUNCTION MID3:REAL

	VAR_INPUT
		IN1 :	REAL;
		IN2 :	REAL;
		IN3 :	REAL;
	END_VAR

	VAR
		_IN1 :	REAL;
		_IN2 :	REAL;
		_IN3 :	REAL;
	END_VAR

	_IN1 := IN1;
	_IN2 := IN2;
	_IN3 := IN3;

	IF _IN1 > _IN2 THEN MID3 := _IN1; _IN1 := _IN2; _IN2 := MID3; END_IF;
	IF _IN2 > _IN3 THEN _IN2 := _IN3; END_IF;
	MID3 := SEL(_IN1 > _IN2, _IN2, _IN1);

END_FUNCTION

PROGRAM program0
	VAR
		IN1 :	REAL;
		IN2 :	REAL;
		IN3 :	REAL;

		OUT : REAL;
	END_VAR

	OUT := MID3(IN1, IN2, IN3);

END_PROGRAM

CONFIGURATION Config0

	RESOURCE Res0 ON PLC
		TASK task0(INTERVAL := T#20ms,PRIORITY := 0);
		PROGRAM instance0 WITH task0 : program0;
	END_RESOURCE

END_CONFIGURATION

(* ---- MIN3.ST ---- *)
FUNCTION MIN3:REAL

	VAR_INPUT
		IN1 :	REAL;
		IN2 :	REAL;
		IN3 :	REAL;
	END_VAR

	MIN3 := MIN(MIN(IN1,IN2),IN3);

END_FUNCTION

PROGRAM program0

	VAR
		IN1 :	REAL;
		IN2 :	REAL;
		IN3 :	REAL;
		CEIL5_OUT : REAL;
	END_VAR

	CEIL5_OUT := MIN3(IN1, IN2, IN3);

END_PROGRAM

CONFIGURATION Config0

	RESOURCE Res0 ON PLC
		TASK task0(INTERVAL := T#20ms,PRIORITY := 0);
		PROGRAM instance0 WITH task0 : program0;
	END_RESOURCE

END_CONFIGURATION

(* ---- MINUTE.ST ---- *)
FUNCTION MINUTE:INT

	VAR_INPUT
		ITOD :	UDINT;
	END_VAR

	minute := UDINT_TO_INT((itod / UDINT#60000) - ((itod / UDINT#3600000) * UDINT#60));

END_FUNCTION

PROGRAM program0
  VAR
	  ITOD :	UDINT;
    CEIL5_OUT : INT;
  END_VAR

  CEIL5_OUT := MINUTE(ITOD);
END_PROGRAM

CONFIGURATION Config0

  RESOURCE Res0 ON PLC
    TASK task0(INTERVAL := T#20ms,PRIORITY := 0);
    PROGRAM instance0 WITH task0 : program0;
  END_RESOURCE
END_CONFIGURATION

(* ---- MINUTE_OF_DT.ST ---- *)
FUNCTION MINUTE_OF_DT:INT
	VAR_INPUT
		XDT :	UDINT;
	END_VAR

	MINUTE_OF_DT := UDINT_TO_INT((XDT MOD UDINT#3600) / UDINT#60);
END_FUNCTION

PROGRAM program0
  VAR
    LocalVar0 : UDINT;
	LocalOUT  : INT;
  END_VAR
  	LocalOUT := MINUTE_OF_DT(LocalVar0);
END_PROGRAM

CONFIGURATION Config0
  RESOURCE Res0 ON PLC
    TASK task0(INTERVAL := T#20ms,PRIORITY := 0);
    PROGRAM instance0 WITH task0 : program0;
  END_RESOURCE
END_CONFIGURATION

(* ---- MINUTE_TO_TIME.ST ---- *)
FUNCTION _REAL_TO_UDINT:UDINT

  	VAR_INPUT
		X :	REAL;
	END_VAR

	IF REAL_TO_UDINT(0.5) = UDINT#1 THEN
		_REAL_TO_UDINT := REAL_TO_UDINT(x);
	ELSIF X > 0.0 THEN
		_REAL_TO_UDINT := REAL_TO_UDINT(x+0.5);
	ELSIF X < 0.0 THEN
		_REAL_TO_UDINT := REAL_TO_UDINT(x-0.5);
	ELSE
		_REAL_TO_UDINT := UDINT#0;
	END_IF;

END_FUNCTION

FUNCTION MINUTE_TO_TIME:TIME

	VAR_INPUT
		IN :	REAL;
	END_VAR

	minute_to_time := UDINT_TO_TIME(_REAL_TO_UDINT(IN * 60000.0));

END_FUNCTION

PROGRAM program0

	VAR
		IN :	REAL;
		CEIL5_OUT : TIME;
	END_VAR

	CEIL5_OUT := MINUTE_TO_TIME(IN);

END_PROGRAM

CONFIGURATION Config0

	RESOURCE Res0 ON PLC
		TASK task0(INTERVAL := T#20ms,PRIORITY := 0);
		PROGRAM instance0 WITH task0 : program0;
	END_RESOURCE

END_CONFIGURATION

(* ---- MIX.ST ---- *)
FUNCTION MIX:REAL

	VAR_INPUT
		A :	REAL;
		B :	REAL;
		M :	REAL;
	END_VAR

	MIX := (1.0 - M) * A + M * B;

END_FUNCTION

PROGRAM program0
	VAR
		A :	REAL;
		B :	REAL;
		M :	REAL;

		OUT : REAL;
	END_VAR

	OUT := MIX(A, B, M);

END_PROGRAM

CONFIGURATION Config0

	RESOURCE Res0 ON PLC
		TASK task0(INTERVAL := T#20ms,PRIORITY := 0);
		PROGRAM instance0 WITH task0 : program0;
	END_RESOURCE

END_CONFIGURATION

(* ---- MODR.ST ---- *)
FUNCTION FLOOR2 : DINT
	VAR_INPUT
		x : REAL;
	END_VAR

	FLOOR2 := REAL_TO_DINT(X);
	IF DINT_TO_REAL(FLOOR2) > X THEN
		FLOOR2 := FLOOR2 - DINT#1;
	END_IF;

END_FUNCTION

FUNCTION MODR: REAL

	VAR_INPUT
		IN :	REAL;
		DIVI :	REAL;
	END_VAR

	IF divi = 0.0 THEN
		MODR := 0.0;
	ELSE
		MODR := in - DINT_TO_REAL(FLOOR2(in / divi)) * divi;
	END_IF;

END_FUNCTION

PROGRAM program0

  	VAR
		IN :	REAL;
		DIVI :	REAL;
		CEIL5_OUT : REAL;
  	END_VAR

  	CEIL5_OUT := MODR(IN, DIVI);
END_PROGRAM

CONFIGURATION Config0

  RESOURCE Res0 ON PLC
    TASK task0(INTERVAL := T#20ms,PRIORITY := 0);
    PROGRAM instance0 WITH task0 : program0;
  END_RESOURCE
END_CONFIGURATION

(* ---- MONTH_BEGIN.ST ---- *)
FUNCTION LEAP_OF_DATE:BOOL

	VAR_INPUT
		IDATE :	UDINT;
	END_VAR

	LEAP_OF_DATE := SHL(UDINT_TO_DWORD((idate + UDINT#43200) / UDINT#31557600), 30) = DWORD#16#80000000;
END_FUNCTION

FUNCTION DAY_OF_YEAR:INT
	VAR_INPUT
		IDATE :	UDINT;
	END_VAR

	DAY_OF_YEAR := UDINT_TO_INT(((idate) / UDINT#86400) MOD UDINT#1461);
	IF DAY_OF_YEAR > 729 THEN
		IF DAY_OF_YEAR > 1095 THEN DAY_OF_YEAR := DAY_OF_YEAR - 1095; ELSE DAY_OF_YEAR := DAY_OF_YEAR - 729; END_IF;
	ELSIF DAY_OF_YEAR > 364 THEN
		DAY_OF_YEAR := DAY_OF_YEAR - 364;
	ELSE
		DAY_OF_YEAR := DAY_OF_YEAR + 1;
	END_IF;
END_FUNCTION

FUNCTION MONTH_OF_DATE:INT

	VAR_INPUT
		IDATE :	UDINT;
	END_VAR

	MONTH_OF_DATE := DAY_OF_YEAR(idate);
	IF MONTH_OF_DATE < 32 THEN
		MONTH_OF_DATE := 1;
	ELSIF LEAP_OF_DATE((IDATE)) THEN
		MONTH_OF_DATE := (MONTH_OF_DATE * 53 + 1668) / 1623;
	ELSE
		MONTH_OF_DATE := (MONTH_OF_DATE * 53 + 1700) / 1620;
	END_IF;
END_FUNCTION

FUNCTION DAY_OF_MONTH:INT
	VAR_INPUT
		IDATE :	UDINT;
	END_VAR

	day_of_month := day_of_year(idate);

	IF leap_of_Date((idate)) THEN
		CASE day_of_month OF
			32..60	:	day_of_month := day_of_month - 31;
			61..91	:	day_of_month := day_of_month - 60;
			92..121 :	day_of_month := day_of_month - 91;
			122..152:	day_of_month := day_of_month - 121;
			153..182:	day_of_month := day_of_month - 152;
			183..213:	day_of_month := day_of_month - 182;
			214..244:	day_of_month := day_of_month - 213;
			245..274:	day_of_month := day_of_month - 244;
			275..305:	day_of_month := day_of_month - 274;
			306..335:	day_of_month := day_of_month - 305;
			336..366:	day_of_month := day_of_month - 335;
		END_CASE;
	ELSE
		CASE day_of_month OF
			32..59	:	day_of_month := day_of_month - 31;
			60..90	:	day_of_month := day_of_month - 59;
			91..120 :	day_of_month := day_of_month - 90;
			121..151:	day_of_month := day_of_month - 120;
			152..181:	day_of_month := day_of_month - 151;
			182..212:	day_of_month := day_of_month - 181;
			213..243:	day_of_month := day_of_month - 212;
			244..273:	day_of_month := day_of_month - 243;
			274..304:	day_of_month := day_of_month - 273;
			305..334:	day_of_month := day_of_month - 304;
			335..365:	day_of_month := day_of_month - 334;
		END_CASE;
	END_IF;
END_FUNCTION

FUNCTION _INT_TO_UDINT:UDINT
	VAR_INPUT
		IN :	INT;
	END_VAR

	_INT_TO_UDINT := DINT_TO_UDINT(INT_TO_DINT(IN));
END_FUNCTION

FUNCTION MONTH_BEGIN:UDINT

VAR_INPUT
	IDATE :	UDINT;
END_VAR

MONTH_BEGIN := idate - _INT_TO_UDINT(DAY_OF_MONTH(idate) - 1) * UDINT#86400;

END_FUNCTION

PROGRAM program0
	VAR
		IDATE :	UDINT;

		OUT : UDINT;
	END_VAR

	OUT := MONTH_BEGIN(IDATE);

END_PROGRAM

CONFIGURATION Config0

	RESOURCE Res0 ON PLC
		TASK task0(INTERVAL := T#20ms,PRIORITY := 0);
		PROGRAM instance0 WITH task0 : program0;
	END_RESOURCE

END_CONFIGURATION

(* ---- MONTH_OF_DATE.ST ---- *)
FUNCTION LEAP_OF_DATE:BOOL

	VAR_INPUT
		IDATE :	UDINT;
	END_VAR

	LEAP_OF_DATE := SHL(UDINT_TO_DWORD((idate + UDINT#43200) / UDINT#31557600), 30) = DWORD#16#80000000;

END_FUNCTION

FUNCTION DAY_OF_YEAR:INT
	VAR_INPUT
		IDATE :	DATE;
	END_VAR

	DAY_OF_YEAR := UDINT_TO_INT((DATE_TO_UDINT(idate) / UDINT#86400) MOD UDINT#1461);
	IF DAY_OF_YEAR > 729 THEN
		IF DAY_OF_YEAR > 1095 THEN DAY_OF_YEAR := DAY_OF_YEAR - 1095; ELSE DAY_OF_YEAR := DAY_OF_YEAR - 729; END_IF;
	ELSIF DAY_OF_YEAR > 364 THEN
		DAY_OF_YEAR := DAY_OF_YEAR - 364;
	ELSE
		DAY_OF_YEAR := DAY_OF_YEAR + 1;
	END_IF;
END_FUNCTION

FUNCTION MONTH_OF_DATE:INT

	VAR_INPUT
		IDATE :	DATE;
	END_VAR

	MONTH_OF_DATE := DAY_OF_YEAR(idate);
	IF MONTH_OF_DATE < 32 THEN
		MONTH_OF_DATE := 1;
	ELSIF LEAP_OF_DATE(DATE_TO_UDINT(IDATE)) THEN
		MONTH_OF_DATE := (MONTH_OF_DATE * 53 + 1668) / 1623;
	ELSE
		MONTH_OF_DATE := (MONTH_OF_DATE * 53 + 1700) / 1620;
	END_IF;

END_FUNCTION

PROGRAM program0
  VAR
    LocalVar0 : DATE;
	LocalOUT  : INT;
  END_VAR
  	LocalOUT := MONTH_OF_DATE(LocalVar0);
END_PROGRAM

CONFIGURATION Config0
  RESOURCE Res0 ON PLC
    TASK task0(INTERVAL := T#20ms,PRIORITY := 0);
    PROGRAM instance0 WITH task0 : program0;
  END_RESOURCE
END_CONFIGURATION

(* ---- MS_TO_BFT.ST ---- *)
FUNCTION MS_TO_BFT:INT

	VAR_INPUT
		MS :	REAL;
	END_VAR

	MS_TO_BFT := REAL_TO_INT(EXPT(MS * 1.196172, 0.666667));

END_FUNCTION

PROGRAM program0
	VAR
		MS :	REAL;

		OUT : INT;
	END_VAR

	OUT := MS_TO_BFT(MS);

END_PROGRAM

CONFIGURATION Config0

	RESOURCE Res0 ON PLC
		TASK task0(INTERVAL := T#20ms,PRIORITY := 0);
		PROGRAM instance0 WITH task0 : program0;
	END_RESOURCE

END_CONFIGURATION

(* ---- MS_TO_KMH.ST ---- *)
FUNCTION MS_TO_KMH:REAL

	VAR_INPUT
		MS :	REAL;
	END_VAR

	MS_TO_KMH := ms * 3.6;

END_FUNCTION

PROGRAM program0
	VAR
		MS :	REAL;

		OUT : REAL;
	END_VAR

	OUT := MS_TO_KMH(MS);

END_PROGRAM

CONFIGURATION Config0

	RESOURCE Res0 ON PLC
		TASK task0(INTERVAL := T#20ms,PRIORITY := 0);
		PROGRAM instance0 WITH task0 : program0;
	END_RESOURCE

END_CONFIGURATION

(* ---- MUL_ADD.ST ---- *)
FUNCTION MUL_ADD:REAL

	VAR_INPUT
		X :	REAL;
		K :	REAL;
		O :	REAL;
	END_VAR

	MUL_ADD := X * K + O;

END_FUNCTION

PROGRAM program0
	VAR
		X :	REAL;
		K :	REAL;
		O :	REAL;

		OUT : REAL;
	END_VAR

	OUT := MUL_ADD(X, K, O);

END_PROGRAM

CONFIGURATION Config0

	RESOURCE Res0 ON PLC
		TASK task0(INTERVAL := T#20ms,PRIORITY := 0);
		PROGRAM instance0 WITH task0 : program0;
	END_RESOURCE

END_CONFIGURATION

(* ---- MULTI_IN.ST ---- *)
FUNCTION MID3:REAL

	VAR_INPUT
		IN1 :	REAL;
		IN2 :	REAL;
		IN3 :	REAL;
	END_VAR

	VAR
		_IN1 :	REAL;
		_IN2 :	REAL;
		_IN3 :	REAL;
	END_VAR

	_IN1 := IN1;
	_IN2 := IN2;
	_IN3 := IN3;

	IF _IN1 > _IN2 THEN MID3 := _IN1; _IN1 := _IN2; _IN2 := MID3; END_IF;
	IF _IN2 > _IN3 THEN _IN2 := _IN3; END_IF;
	MID3 := SEL(_IN1 > _IN2, _IN2, _IN1);

END_FUNCTION

FUNCTION _BYTE_TO_INT:INT
	VAR_INPUT
		IN :	BYTE;
	END_VAR

	_BYTE_TO_INT := USINT_TO_INT(BYTE_TO_USINT(IN));
END_FUNCTION

FUNCTION MULTI_IN:REAL

	VAR_INPUT
		IN_1 :	REAL;
		IN_2 :	REAL;
		IN_3 :	REAL;
		DEFAULT :	REAL;
		IN_MIN :	REAL;
		IN_MAX :	REAL;
		MODE :	BYTE;
	END_VAR

	VAR
		count :	INT;
		F1 :	BOOL;
		F2 :	BOOL;
		F3 :	BOOL;
	END_VAR

	F1 :=  in_1 > in_min AND in_1 < in_max;
	F2 :=  in_2 > in_min AND in_2 < in_max;
	F3 :=  in_3 > in_min AND in_3 < in_max;

	CASE _BYTE_TO_INT(mode) OF
	0:	count := 0;
		IF F1 THEN
			count := count + 1;
			MULTI_IN := in_1;
		ELSE
			MULTI_IN := 0.0;
		END_IF;
		IF F2 THEN
			count := count + 1;
			MULTI_IN := MULTI_IN + in_2;
		END_IF;
		IF F3 THEN
			count := count + 1;
			MULTI_IN := MULTI_IN + in_3;
		END_IF;
		MULTI_IN := SEL_REAL(count = 0, MULTI_IN / INT_TO_REAL(count), default);

	1:	MULTI_IN := SEL_REAL(F1, default, IN_1);

	2:	MULTI_IN := SEL_REAL(F2, default, IN_2);

	3:	MULTI_IN := SEL_REAL(F3, default, IN_3);

	4:	MULTI_IN := default;

	5:	MULTI_IN := SEL_REAL(F1, in_max, IN_1);
		IF F2 AND in_2 < MULTI_IN THEN MULTI_IN := in_2; END_IF;
		IF F3 AND in_3 < MULTI_IN THEN MULTI_IN := in_3; END_IF;
		IF MULTI_IN = in_max THEN MULTI_IN := default; END_IF;

	6:	MULTI_IN := SEL_REAL(F1, in_min, IN_1);
		IF F2 AND in_2 > MULTI_IN THEN MULTI_IN := in_2; END_IF;
		IF F3 AND in_3 > MULTI_IN THEN MULTI_IN := in_3; END_IF;
		IF MULTI_IN = in_min THEN MULTI_IN := default; END_IF;

	7:	IF F1 AND F2 AND F3 THEN MULTI_IN := MID3(in_1, in_2, in_3);
		ELSIF F1 AND F2 THEN MULTI_IN := MIN(in_1, in_2);
		ELSIF F1 AND F3 THEN MULTI_IN := MIN(in_1, in_3);
		ELSIF F2 AND F3 THEN MULTI_IN := MIN(in_2, in_3);
		ELSIF F1 THEN MULTI_IN := in_1;
		ELSIF F2 THEN MULTI_IN := in_2;
		ELSIF F3 THEN MULTI_IN := in_3;
		ELSE MULTI_IN := default;
		END_IF;

	END_CASE;

END_FUNCTION

PROGRAM program0
	VAR
		IN_1 :	REAL;
		IN_2 :	REAL;
		IN_3 :	REAL;
		DEFAULT :	REAL;
		IN_MIN :	REAL;
		IN_MAX :	REAL;
		MODE :	BYTE;

		OUT : REAL;
	END_VAR

	OUT := MULTI_IN(IN_1, IN_2, IN_3, DEFAULT, IN_MIN, IN_MAX, MODE);

END_PROGRAM

CONFIGURATION Config0

	RESOURCE Res0 ON PLC
		TASK task0(INTERVAL := T#20ms,PRIORITY := 0);
		PROGRAM instance0 WITH task0 : program0;
	END_RESOURCE

END_CONFIGURATION

(* ---- MULTIME.ST ---- *)
FUNCTION _REAL_TO_DWORD: DWORD

  VAR_INPUT
    X :	REAL;
  END_VAR

  IF REAL_TO_DWORD(0.5) = DWORD#1 THEN
    _REAL_TO_DWORD := REAL_TO_DWORD(x);
  ELSIF X > 0.0 THEN
    _REAL_TO_DWORD := REAL_TO_DWORD(x+0.5);
  ELSIF X < 0.0 THEN
    _REAL_TO_DWORD := REAL_TO_DWORD(x-0.5);
  ELSE
    _REAL_TO_DWORD := DWORD#0;
  END_IF;
END_FUNCTION

FUNCTION _DWORD_TO_REAL:REAL
	VAR_INPUT
		IN :	DWORD;
	END_VAR

	_DWORD_TO_REAL := UDINT_TO_REAL(DWORD_TO_UDINT(IN));

END_FUNCTION

FUNCTION MULTIME:TIME
	VAR_INPUT
		T :	TIME;
		M :	REAL;
	END_VAR

	multime := DWORD_TO_TIME(_REAL_TO_DWORD(_DWORD_TO_REAL(TIME_TO_DWORD(t))*M));
END_FUNCTION

PROGRAM program0
  VAR
    LocalVar0 : TIME;
	LocalVar1 : REAL;
	LocalOUT  : TIME;
  END_VAR
  	LocalOUT := MULTIME(LocalVar0, LocalVar1);
END_PROGRAM

CONFIGURATION Config0
  RESOURCE Res0 ON PLC
    TASK task0(INTERVAL := T#20ms,PRIORITY := 0);
    PROGRAM instance0 WITH task0 : program0;
  END_RESOURCE
END_CONFIGURATION

(* ---- MUX_2.ST ---- *)
FUNCTION MUX_2:BOOL

	VAR_INPUT
		D0 :	BOOL;
		D1 :	BOOL;
		A0 :	BOOL;
	END_VAR

	MUX_2 := SEL(A0, D0, D1);

END_FUNCTION

PROGRAM program0
	VAR
		D0 :	BOOL;
		D1 :	BOOL;
		A0 :	BOOL;
		OUT : BOOL;
	END_VAR

	OUT := MUX_2(D0, D1, A0);

END_PROGRAM

CONFIGURATION Config0

	RESOURCE Res0 ON PLC
		TASK task0(INTERVAL := T#20ms,PRIORITY := 0);
		PROGRAM instance0 WITH task0 : program0;
	END_RESOURCE

END_CONFIGURATION

(* ---- MUX_4.ST ---- *)
FUNCTION MUX_4:BOOL

	VAR_INPUT
		D0 :	BOOL;
		D1 :	BOOL;
		D2 :	BOOL;
		D3 :	BOOL;
		A0 :	BOOL;
		A1 :	BOOL;
	END_VAR

	IF A1 THEN
		MUX_4 := SEL(A0, D2, D3);
	ELSE
		MUX_4 := SEL(A0, D0, D1);
	END_IF;

END_FUNCTION

PROGRAM program0
	VAR
		D0 :	BOOL;
		D1 :	BOOL;
		D2 :	BOOL;
		D3 :	BOOL;
		A0 :	BOOL;
		A1 :	BOOL;

		OUT : BOOL;
	END_VAR

	OUT := MUX_4(D0, D1, D2, D3, A0, A1);

END_PROGRAM

CONFIGURATION Config0

	RESOURCE Res0 ON PLC
		TASK task0(INTERVAL := T#20ms,PRIORITY := 0);
		PROGRAM instance0 WITH task0 : program0;
	END_RESOURCE

END_CONFIGURATION

(* ---- MUX_R2.ST ---- *)
FUNCTION MUX_R2:REAL

	VAR_INPUT
		IN0 :	REAL;
		IN1 :	REAL;
		A :	BOOL;
	END_VAR

	MUX_R2 := SEL(A, IN0, IN1);

END_FUNCTION

PROGRAM program0
	VAR
		IN0 :	REAL;
		IN1 :	REAL;
		A :	BOOL;

		OUT : REAL;
	END_VAR

	OUT := MUX_R2(IN0, IN1, A);

END_PROGRAM

CONFIGURATION Config0

	RESOURCE Res0 ON PLC
		TASK task0(INTERVAL := T#20ms,PRIORITY := 0);
		PROGRAM instance0 WITH task0 : program0;
	END_RESOURCE

END_CONFIGURATION

(* ---- MUX_R4.ST ---- *)
FUNCTION MUX_R4:REAL

	VAR_INPUT
		IN0 :	REAL;
		IN1 :	REAL;
		IN2 :	REAL;
		IN3 :	REAL;
		A0 :	BOOL;
		A1 :	BOOL;
	END_VAR

	IF A1 THEN
		MUX_R4 := SEL(A0, IN2, IN3);
	ELSE
		MUX_R4 := SEL(A0, IN0, IN1);
	END_IF;

END_FUNCTION

PROGRAM program0
	VAR
		IN0 :	REAL;
		IN1 :	REAL;
		IN2 :	REAL;
		IN3 :	REAL;
		A0 :	BOOL;
		A1 :	BOOL;

		OUT : REAL;
	END_VAR

	OUT := MUX_R4(IN0, IN1, IN2, IN3, A0, A1);

END_PROGRAM

CONFIGURATION Config0

	RESOURCE Res0 ON PLC
		TASK task0(INTERVAL := T#20ms,PRIORITY := 0);
		PROGRAM instance0 WITH task0 : program0;
	END_RESOURCE

END_CONFIGURATION

(* ---- NEGX.ST ---- *)
FUNCTION NEGX:REAL

	VAR_INPUT
		X :	REAL;
	END_VAR

	NEGX := -X;

END_FUNCTION

PROGRAM program0
	VAR
		_X : REAL;
		OUT : REAL;
	END_VAR

	OUT := NEGX(_X);
END_PROGRAM

CONFIGURATION Config0

	RESOURCE Res0 ON PLC
		TASK task0(INTERVAL := T#20ms,PRIORITY := 0);
		PROGRAM instance0 WITH task0 : program0;
	END_RESOURCE

END_CONFIGURATION

(* ---- NETWORK_VERSION.ST ---- *)
FUNCTION _INT_TO_UDINT:UDINT
	VAR_INPUT
		IN :	INT;
	END_VAR

	_INT_TO_UDINT := DINT_TO_UDINT(INT_TO_DINT(IN));
END_FUNCTION

FUNCTION SET_DATE:UDINT

	VAR_INPUT
		YEAR :	INT;
		MONTH :	INT;
		DAY :	INT;
	END_VAR

	VAR
		count :	INT;
	END_VAR

	IF month > 2 THEN
		count := (month - 1) * 30;
		IF month > 7 THEN
			count := count + DWORD_TO_INT(SHR(DINT_TO_DWORD(INT_TO_DINT(month) - INT_TO_DINT(3)),1));
		ELSE
			count := count + DWORD_TO_INT(SHR(DINT_TO_DWORD(INT_TO_DINT(month) - INT_TO_DINT(4)),1));
		END_IF;
		IF SHL(INT_TO_WORD(year),14) = WORD#0 THEN
			count := count + 1;
		END_IF;
	ELSE
		count := (month - 1) * 31;
	END_IF;
	SET_DATE := (_INT_TO_UDINT(count + day - 1) + DWORD_TO_UDINT(SHR(UDINT_TO_DWORD(_INT_TO_UDINT(year) * UDINT#1461 - UDINT#2878169), 2))) * UDINT#86400;

END_FUNCTION

FUNCTION NETWORK_VERSION:DWORD

	VAR_INPUT
		IN :	BOOL;
	END_VAR

	IF in THEN
		NETWORK_VERSION := UDINT_TO_DWORD(set_Date(2011,12,01));
	ELSE
		NETWORK_VERSION := DWORD#121;
	END_IF;

END_FUNCTION

PROGRAM program0
	VAR
		IN :	BOOL;
		CEIL5_OUT : DWORD;
	END_VAR

  	CEIL5_OUT := NETWORK_VERSION(IN);
END_PROGRAM

CONFIGURATION Config0

  RESOURCE Res0 ON PLC
    TASK task0(INTERVAL := T#20ms,PRIORITY := 0);
    PROGRAM instance0 WITH task0 : program0;
  END_RESOURCE
END_CONFIGURATION

(* ---- OFFSET.ST ---- *)
FUNCTION _OFFSET:REAL

	VAR_INPUT
		X :	REAL;
		O1 :	BOOL;
		O2 :	BOOL;
		O3 :	BOOL;
		O4 :	BOOL;
		D :	BOOL;
		OFFSET_1 :	REAL;
		OFFSET_2 :	REAL;
		OFFSET_3 :	REAL;
		OFFSET_4 :	REAL;
		DEFAULT :	REAL;
	END_VAR

	IF D THEN _Offset := default; ELSE _Offset := X; END_IF;
	IF O1 THEN _Offset := _Offset + offset_1; END_IF;
	IF O2 THEN _Offset := _Offset + offset_2; END_IF;
	IF O3 THEN _Offset := _Offset + offset_3; END_IF;
	IF O4 THEN _Offset := _Offset + offset_4; END_IF;

END_FUNCTION

PROGRAM program0

	VAR
		X :	REAL;
		O1 :	BOOL;
		O2 :	BOOL;
		O3 :	BOOL;
		O4 :	BOOL;
		D :	BOOL;
		OFFSET_1 :	REAL;
		OFFSET_2 :	REAL;
		OFFSET_3 :	REAL;
		OFFSET_4 :	REAL;
		DEFAULT :	REAL;
		OUT : REAL;
	END_VAR

	OUT := _OFFSET(X, O1, O2, O3, O4, D, OFFSET_1, OFFSET_2, OFFSET_3, OFFSET_4, DEFAULT);
END_PROGRAM

CONFIGURATION Config0

	RESOURCE Res0 ON PLC
		TASK task0(INTERVAL := T#20ms,PRIORITY := 0);
		PROGRAM instance0 WITH task0 : program0;
	END_RESOURCE

END_CONFIGURATION

(* ---- OFFSET2.ST ---- *)
FUNCTION OFFSET2:REAL

	VAR_INPUT
		X :	REAL;
		O1 :	BOOL;
		O2 :	BOOL;
		O3 :	BOOL;
		O4 :	BOOL;
		D :	BOOL;
		OFFSET_1 :	REAL;
		OFFSET_2 :	REAL;
		OFFSET_3 :	REAL;
		OFFSET_4 :	REAL;
		DEFAULT :	REAL;
	END_VAR

	IF D THEN Offset2 := default; ELSE Offset2 := X; END_IF;
	IF O4 THEN Offset2 := Offset2 + offset_4;
	ELSIF O3 THEN Offset2 := Offset2 + offset_3;
	ELSIF O2 THEN Offset2 := Offset2 + offset_2;
	ELSIF O1 THEN Offset2 := Offset2 + offset_1;
	END_IF;

END_FUNCTION

PROGRAM program0
	VAR
		X :	REAL;
		O1 :	BOOL;
		O2 :	BOOL;
		O3 :	BOOL;
		O4 :	BOOL;
		D :	BOOL;
		OFFSET_1 :	REAL;
		OFFSET_2 :	REAL;
		OFFSET_3 :	REAL;
		OFFSET_4 :	REAL;
		DEFAULT :	REAL;
		OUT : REAL;
	END_VAR

	OUT := OFFSET2(X, O1, O2, O3, O4, D, OFFSET_1, OFFSET_2, OFFSET_3, OFFSET_4, DEFAULT);
END_PROGRAM

CONFIGURATION Config0

	RESOURCE Res0 ON PLC
		TASK task0(INTERVAL := T#20ms,PRIORITY := 0);
		PROGRAM instance0 WITH task0 : program0;
	END_RESOURCE

END_CONFIGURATION

(* ---- OM_TO_F.ST ---- *)
FUNCTION OM_TO_F:REAL

	VAR_INPUT
		OM :	REAL;
	END_VAR

	OM_to_F := OM / 6.283185307179586476;

END_FUNCTION

PROGRAM program0
	VAR
		OM : REAL;
		OUT : REAL;
	END_VAR

	OUT := OM_TO_F(OM);
END_PROGRAM

CONFIGURATION Config0

	RESOURCE Res0 ON PLC
		TASK task0(INTERVAL := T#20ms,PRIORITY := 0);
		PROGRAM instance0 WITH task0 : program0;
	END_RESOURCE

END_CONFIGURATION

(* ---- OSCAT_VERSION.ST ---- *)
FUNCTION _INT_TO_UDINT:UDINT
	VAR_INPUT
		IN :	INT;
	END_VAR

	_INT_TO_UDINT := DINT_TO_UDINT(INT_TO_DINT(IN));
END_FUNCTION

FUNCTION SET_DATE:UDINT

	VAR_INPUT
		YEAR :	INT;
		MONTH :	INT;
		DAY :	INT;
	END_VAR

	VAR
		count :	INT;
	END_VAR

	IF month > 2 THEN
		count := (month - 1) * 30;
		IF month > 7 THEN
			count := count + DWORD_TO_INT(SHR(DINT_TO_DWORD(INT_TO_DINT(month) - INT_TO_DINT(3)),1));
		ELSE
			count := count + DWORD_TO_INT(SHR(DINT_TO_DWORD(INT_TO_DINT(month) - INT_TO_DINT(4)),1));
		END_IF;
		IF SHL(INT_TO_WORD(year),14) = WORD#0 THEN
			count := count + 1;
		END_IF;
	ELSE
		count := (month - 1) * 31;
	END_IF;
	SET_DATE := (_INT_TO_UDINT(count + day - 1) + DWORD_TO_UDINT(SHR(UDINT_TO_DWORD(_INT_TO_UDINT(year) * UDINT#1461 - UDINT#2878169), 2))) * UDINT#86400;

END_FUNCTION

FUNCTION OSCAT_VERSION:DWORD

	VAR_INPUT
		IN :	BOOL;
	END_VAR

	IF in THEN
		Oscat_version := UDINT_TO_DWORD(set_Date(2012,01,02));
	ELSE
		Oscat_version := DWORD#333;
	END_IF;

END_FUNCTION

PROGRAM program0
	VAR
		IN :	BOOL;
		OUT : DWORD;
	END_VAR

	OUT := OSCAT_VERSION(IN);
END_PROGRAM

CONFIGURATION Config0

	RESOURCE Res0 ON PLC
		TASK task0(INTERVAL := T#20ms,PRIORITY := 0);
		PROGRAM instance0 WITH task0 : program0;
	END_RESOURCE

END_CONFIGURATION

(* ---- PARITY.ST ---- *)
FUNCTION BIT_OF_DWORD : BOOL

	VAR_INPUT
		IN : DWORD;
		N : INT;
	END_VAR

	BIT_OF_DWORD := (SHR(in,N) AND 16#00000001) > 0;

END_FUNCTION

FUNCTION PARITY:BOOL

	VAR_INPUT
		IN :	DWORD;
	END_VAR

	VAR
		in2 :	DWORD;
	END_VAR

	in2:=in;
	WHILE in2 > DWORD#0 DO
		parity := parity XOR BIT_OF_DWORD(in2,0) XOR BIT_OF_DWORD(in2,1) XOR BIT_OF_DWORD(in2,2) XOR BIT_OF_DWORD(in2,3);
		in2 := SHR(in2,4);
	END_WHILE;

END_FUNCTION

PROGRAM program0
	VAR
		IN : DWORD;
		OUT : BOOL;
	END_VAR

	OUT := PARITY(IN);
END_PROGRAM

CONFIGURATION Config0

	RESOURCE Res0 ON PLC
		TASK task0(INTERVAL := T#20ms,PRIORITY := 0);
		PROGRAM instance0 WITH task0 : program0;
	END_RESOURCE

END_CONFIGURATION

(* ---- PERIOD.ST ---- *)
FUNCTION LEAP_OF_DATE:BOOL

	VAR_INPUT
		IDATE :	UDINT;
	END_VAR

	LEAP_OF_DATE := SHL(UDINT_TO_DWORD((idate + UDINT#43200) / UDINT#31557600), 30) = DWORD#16#80000000;
END_FUNCTION

FUNCTION DAY_OF_YEAR:INT
	VAR_INPUT
		IDATE :	UDINT;
	END_VAR

	DAY_OF_YEAR := UDINT_TO_INT(((idate) / UDINT#86400) MOD UDINT#1461);
	IF DAY_OF_YEAR > 729 THEN
		IF DAY_OF_YEAR > 1095 THEN DAY_OF_YEAR := DAY_OF_YEAR - 1095; ELSE DAY_OF_YEAR := DAY_OF_YEAR - 729; END_IF;
	ELSIF DAY_OF_YEAR > 364 THEN
		DAY_OF_YEAR := DAY_OF_YEAR - 364;
	ELSE
		DAY_OF_YEAR := DAY_OF_YEAR + 1;
	END_IF;
END_FUNCTION

FUNCTION PERIOD:BOOL

	VAR
		day1 :	INT;
		day2 :	INT;
		dayx :	INT;
	END_VAR

	VAR_INPUT
		D1 :	UDINT;
		Dx :	UDINT;
		D2 :	UDINT;
	END_VAR

	day1 := day_of_year(d1);
	day2 := day_of_year(d2);
	dayx := day_of_year(dx);
	IF NOT leap_of_Date(dx) AND dayx > 58 THEN dayx := dayx + 1; END_IF;
	IF NOT leap_of_Date(d1) AND day1 > 58 THEN day1 := day1 + 1; END_IF;
	IF NOT leap_of_Date(d2) AND day2 > 58 THEN day2 := day2 + 1; END_IF;

	IF day2 < day1 THEN
		(* the period spans over the new year *)
		period := dayx <= day2 OR dayx >= day1;
	ELSE
		period := dayx >= day1 AND dayx <= day2;
	END_IF;

END_FUNCTION

PROGRAM program0
	VAR
		D1 :	UDINT;
		Dx :	UDINT;
		D2 :	UDINT;

		OUT : BOOL;
	END_VAR

	OUT := PERIOD(D1, Dx, D2);
END_PROGRAM

CONFIGURATION Config0

	RESOURCE Res0 ON PLC
		TASK task0(INTERVAL := T#20ms,PRIORITY := 0);
		PROGRAM instance0 WITH task0 : program0;
	END_RESOURCE

END_CONFIGURATION

(* ---- PT_TO_F.ST ---- *)
FUNCTION _DWORD_TO_REAL:REAL
	VAR_INPUT
		IN :	DWORD;
	END_VAR

	_DWORD_TO_REAL := UDINT_TO_REAL(DWORD_TO_UDINT(IN));

END_FUNCTION

FUNCTION PT_TO_F:REAL

	VAR_INPUT
		PT :	TIME;
	END_VAR

	PT_TO_F := 1000.0 / _DWORD_TO_REAL(TIME_TO_DWORD(PT));

END_FUNCTION

PROGRAM program0
  VAR
    PT : TIME;
    OUT : REAL;
  END_VAR

  OUT := PT_TO_F(PT);
END_PROGRAM

CONFIGURATION Config0

  RESOURCE Res0 ON PLC
    TASK task0(INTERVAL := T#20ms,PRIORITY := 0);
    PROGRAM instance0 WITH task0 : program0;
  END_RESOURCE
END_CONFIGURATION

(* ---- RAD.ST ---- *)
FUNCTION FLOOR2 : DINT
	VAR_INPUT
		x : REAL;
	END_VAR

	FLOOR2 := REAL_TO_DINT(X);
	IF DINT_TO_REAL(FLOOR2) > X THEN
		FLOOR2 := FLOOR2 - DINT#1;
	END_IF;

END_FUNCTION

FUNCTION MODR: REAL

	VAR_INPUT
		IN :	REAL;
		DIVI :	REAL;
	END_VAR

	IF divi = 0.0 THEN
		MODR := 0.0;
	ELSE
		MODR := in - DINT_TO_REAL(FLOOR2(in / divi)) * divi;
	END_IF;

END_FUNCTION

FUNCTION RAD:REAL

	VAR_INPUT
		DEG :	REAL;
	END_VAR

	RAD := MODR(0.0174532925199433 * DEG , 6.283185307179586476);

END_FUNCTION

PROGRAM program0

	VAR
		DEG :	REAL;
		CEIL5_OUT : REAL;
	END_VAR

	CEIL5_OUT := RAD(DEG);

END_PROGRAM

CONFIGURATION Config0

	RESOURCE Res0 ON PLC
		TASK task0(INTERVAL := T#20ms,PRIORITY := 0);
		PROGRAM instance0 WITH task0 : program0;
	END_RESOURCE

END_CONFIGURATION

(* ---- RANGE_TO_BYTE.ST ---- *)
FUNCTION TRUNC_REAL:REAL

	VAR_INPUT
		IN :	REAL;
	END_VAR

	TRUNC_REAL := UDINT_TO_REAL(DINT_TO_UDINT(TRUNC(IN)));
END_FUNCTION

FUNCTION RANGE_TO_BYTE:BYTE

	VAR_INPUT
		X :	REAL;
		LOW :	REAL;
		HIGH :	REAL;
	END_VAR

	Range_to_Byte := REAL_TO_BYTE(TRUNC_REAL((LIMIT(low,X,high)-low) * 255.0 / (high - low)));

END_FUNCTION

PROGRAM program0

	VAR
		X :	REAL;
		LOW :	REAL;
		HIGH :	REAL;

        OUT :	BYTE;
	END_VAR
	OUT := RANGE_TO_BYTE(X, LOW, HIGH);

END_PROGRAM

CONFIGURATION Config0

	RESOURCE Res0 ON PLC
		TASK task0(INTERVAL := T#20ms,PRIORITY := 0);
		PROGRAM instance0 WITH task0 : program0;
	END_RESOURCE

END_CONFIGURATION

(* ---- RANGE_TO_WORD.ST ---- *)
FUNCTION TRUNC_REAL:REAL

	VAR_INPUT
		IN :	REAL;
	END_VAR

	TRUNC_REAL := UDINT_TO_REAL(DINT_TO_UDINT(TRUNC(IN)));
END_FUNCTION

FUNCTION RANGE_TO_WORD:WORD

	VAR_INPUT
		X :	REAL;
		LOW :	REAL;
		HIGH :	REAL;
	END_VAR

	Range_to_Word := REAL_TO_WORD(TRUNC_REAL((LIMIT(low,X,high)-low) * 65535.0 / (high - low)));

END_FUNCTION

PROGRAM program0

	VAR
		X :	REAL;
		LOW :	REAL;
		HIGH :	REAL;

        OUT :	WORD;
	END_VAR
	OUT := RANGE_TO_WORD(X, LOW, HIGH);

END_PROGRAM

CONFIGURATION Config0

	RESOURCE Res0 ON PLC
		TASK task0(INTERVAL := T#20ms,PRIORITY := 0);
		PROGRAM instance0 WITH task0 : program0;
	END_RESOURCE

END_CONFIGURATION

(* ---- REAL_TO_TIME.ST ---- *)
FUNCTION _REAL_TO_UDINT:UDINT
  VAR_INPUT
    X :	REAL;
  END_VAR

  IF REAL_TO_UDINT(0.5) = UDINT#1 THEN
    _REAL_TO_UDINT := REAL_TO_UDINT(x);
  ELSIF X > 0.0 THEN
    _REAL_TO_UDINT := REAL_TO_UDINT(x+0.5);
  ELSIF X < 0.0 THEN
    _REAL_TO_UDINT := REAL_TO_UDINT(x-0.5);
  ELSE
    _REAL_TO_UDINT := UDINT#0;
  END_IF;
END_FUNCTION

FUNCTION REAL_TO_TIME2:TIME
	VAR_INPUT
		IN :	REAL;
	END_VAR

	REAL_TO_TIME2 := DINT_TO_TIME(UDINT_TO_DINT(_REAL_TO_UDINT(IN)));
END_FUNCTION

PROGRAM program0
  VAR
    LocalVar0 : REAL;
    LocalOUT  : TIME;
  END_VAR

  LocalOUT := REAL_TO_TIME2(LocalVar0);
END_PROGRAM

CONFIGURATION Config0
  RESOURCE Res0 ON PLC
    TASK task0(INTERVAL := T#20ms,PRIORITY := 0);
    PROGRAM instance0 WITH task0 : program0;
  END_RESOURCE
END_CONFIGURATION

(* ---- REFLECT.ST ---- *)
FUNCTION REFLECT:DWORD
	VAR_INPUT
		D :	DWORD;
		L :	INT;
	END_VAR

	VAR
		i :	INT;
		_d :	DWORD;
	END_VAR

	REFLECT := DWORD#0;
	_d := D;
	FOR i := 1 TO L DO
		REFLECT := SHL(REFLECT, 1) OR BOOL_TO_DWORD((_d AND DWORD#2#0000_0001) > DWORD#0); (* D.0 *)
		_d := SHR(_d, 1);
	END_FOR;
	REFLECT := REFLECT OR SHL(_d, L);
END_FUNCTION

PROGRAM program0
  VAR
    LocalVar0 : DWORD;
	LocalVar1 : INT;
	LocalOUT  : DWORD;
  END_VAR
  	LocalOUT := REFLECT(LocalVar0, LocalVar1);
END_PROGRAM

CONFIGURATION Config0
  RESOURCE Res0 ON PLC
    TASK task0(INTERVAL := T#20ms,PRIORITY := 0);
    PROGRAM instance0 WITH task0 : program0;
  END_RESOURCE
END_CONFIGURATION

(* ---- REFRACTION.ST ---- *)
FUNCTION REFRACTION:REAL

	VAR_INPUT
		ELEV :	REAL;
	END_VAR

	VAR
		tmp :	REAL;
	END_VAR

	tmp := LIMIT(-1.9, elev, 80.0);
	REFRACTION := 0.0174532925199433 / TAN(0.0174532925199433 * (tmp + 10.3 / (tmp + 5.11)));

END_FUNCTION

PROGRAM program0

	VAR
		ELEV :	REAL;

		OUT :	REAL;
	END_VAR
	OUT := REFRACTION(ELEV);

END_PROGRAM

CONFIGURATION Config0

	RESOURCE Res0 ON PLC
		TASK task0(INTERVAL := T#20ms,PRIORITY := 0);
		PROGRAM instance0 WITH task0 : program0;
	END_RESOURCE

END_CONFIGURATION
